TYPE "IOL_CONF"
// stored: IsFailsafeCompliant false
   STRUCT
      SELECTED : Struct
         SCRN_1 : Bool;   // SCREEN ONE SELECTED / SCREEN 1 SELECTED
         SCRN_2 : Bool;   // SCREEN TWO SELECTED / SCREEN 2 SELECTED
         SCRN_3 : Bool;   // SCREEN THREE SELECTED / SCREEN 3 SELECTED
         SCRN_4 : Bool;   // SCREEN FOUR SELECTED / SCREEN 4 SELECTED
         SCRN_5 : Bool;   // SCREEN FIVE SELECTED / SCREEN 5 SELECTED
         SCRN_6 : Bool;   // SCREEN SIX SELECTED / SCREEN 6 SELECTED
         SCRN_7 : Bool;   // SCREEN SEVEN SELECTED / SCREEN 7 SELECTED
         SCRN_8 : Bool;   // SCREEN EIGHT SELECTED / SCREEN 8 SELECTED
         SCRN_11 : Bool;   // SCREEN 11 SELECTED
         SCRN_12 : Bool;   // SCREEN 12 SELECTED
         SCRN_13 : Bool;   // SCREEN 13 SELECTED
         SCRN_14 : Bool;   // SCREEN 14 SELECTED
         SCRN_15 : Bool;   // SCREEN 15 SELECTED
         SCRN_16 : Bool;   // SCREEN 16 SELECTED
         SCRN_17 : Bool;   // SCREEN 17 SELECTED
         SCRN_18 : Bool;   // SCREEN 18 SELECTED
      END_STRUCT;
      HMI_VARIABLES : Struct
         DONE : Bool;   // HMI DONE BIT
         BUSY : Bool;   // HMI BUSY BIT
         ERROR : Bool;   // HMI ERROR BIT
         RD_WRT_HMI : Bool;   // HMI BUTTON READ/ WRITE SELECTION
         EXECUTE_ACTION : Bool;   // HMI EXECUTE READ/WRITE
         SPARE_205 : Bool;   // SPARE BIT
         SPARE_206 : Bool;   // SPARE BIT
         SPARE_207 : Bool;   // SPARE BIT
         SPARE_210 : Bool;   // SPARE BIT
         SPARE_211 : Bool;   // SPARE BIT
         SPARE_212 : Bool;   // SPARE BIT
         SPARE_213 : Bool;   // SPARE BIT
         SPARE_214 : Bool;   // SPARE BIT
         SPARE_215 : Bool;   // SPARE BIT
         SPARE_216 : Bool;   // SPARE BIT
         SPARE_217 : Bool;   // SPARE BIT
         IOL_LIST : Int;   // SELECTION LIST
         IO_LIST_OLD : Int;   // SELECTION LIST OLD
         SCRN_NMBR : Int;   // SELECTED SCREEN
         SCRN_NMBR_OLD : Int;   // SELECTED SCREEN OLD
         RND_INTRVL_1 : Real;   // ROUND INTERVAL FIRST VALUE
         RND_INTRVL_2 : Real;   // ROUND INTVERAL SECOND VALUE
         VAR_ERROR : Byte;   // VARIABLE NUMBER ERROR TAKE PLACE
         TOT_FLT : Byte;   // TOTAL FAULT
         FIRST_VALUE_DISPLAY : Real;   // HMI FIRST VALUE DISPLAY
         SECOND_VALUE_DISPLAY : Real;   // HMI SECOND VALUE DISPLAY
         SPARE_DISPLAY0 : Real;   // HMI SPARE DISPLAY
         SPARE_DISPLAY1 : Real;   // HMI SPARE DISPLAY
         SPARE_DISPLAY2 : Real;   // HMI SPARE DISPLAY
         REAL_VALUE : Array[0..17] of Real;   // REAL VALUE
      END_STRUCT;
      SPARE : Array[1..24] of Byte;
      GEOADR { ExternalAccessible := 'False'; ExternalVisible := 'False'; ExternalWritable := 'False'; S7_SetPoint := 'True'} : GEOADDR;   // INFO TO DETERMINE HW_IO
      CONFIG_DATA : Struct
         SPARE : UInt;   // DATA ADDRESS ID / Spare
         DATA_PORT : UInt;   // DATA PORT
         CAP_NMBR : UInt;   // CAP NUMBER
         VAR_RO : UInt;   // READ ONLY VARIABLES
         TOT_REAL_VAR : UInt;   // TOTAL REAL VARIABLES TO READ
         REAL_VAR_ARRAY_POS : UInt;   // REAL VARIABLES FIRST POSITION AT ARRAY
         TOT_VAR_TO_RD : UInt;   // TOTAL VARIABLES TO READ
      END_STRUCT;
      IOL_CONF : Array[1..20] of Struct
         INDX : Int;   // INDEX
         SBINDX : Int;   // SUBINDEX
         LNG : Int;   // LENGTH
         GRDNT : Real;   // GRADIENT
         OFFST : Real;   // OFFSET
         ROUND_1_OR_2 : Int;   // ROUND INTERVAL TO USE 1 OR 2
      END_STRUCT;
   END_STRUCT;
   // // GEOADR.HWTYPE : HW type (info to obtain from hw component) 4=module
   // // GEOADR.AREA : Normally not used
   // // GEOADR.IOSYSTEM : Network the IO master is on (100 profinet)(Normally always 100)
   // // GEOADR.STATION : Device No. of the IO master in hardware
   // // GEOADR.SLOT : Slot Number in hardware
   // // GEOADR.SUBSLOT : Sub Slot Number if necessary (Normally not used)
END_TYPE

TYPE "LIOLink_typeDiagnostics"
// stored: IsFailsafeCompliant false
   STRUCT
      status { ExternalVisible := 'False'; ExternalWritable := 'False'} : Word;   // Status of the Block or error identification when error occurred
      subfunctionStatus { ExternalVisible := 'False'; ExternalWritable := 'False'} : DWord;   // Status or return value of called FB's, FCs and system blocks
      stateNumber { ExternalVisible := 'False'; ExternalWritable := 'False'} : DInt;   // State in the state machine of the block where the error occurred
   END_STRUCT;
END_TYPE

TYPE "AXIS_MANAGEMENT"
// stored: IsFailsafeCompliant false
   STRUCT
      UNIT_01_HM_PSTN : Bool;   // UNIT 01 HOME POSITION
      UNIT_01_MAINT_POS : Bool;   // UNIT 01 MAINTENACE POSITION
      UNIT_01_ST1_OUT_OF_CLLSN_ST0 : Bool;   // UNIT 01 STATION 1 OUT OF COLLISION STATION 0
      UNIT_01_ST2_OUT_OF_CLLSN_ST0 : Bool;   // UNIT 01 STATION 2 OUT OF COLLISION STATION 0
      UNIT_01_ST3_OUT_OF_CLLSN_ST0 : Bool;   // UNIT 01 STATION 3 OUT OF COLLISION STATION 0
      UNIT_01_ST4_OUT_OF_CLLSN_ST0 : Bool;   // UNIT 01 STATION 4 OUT OF COLLISION STATION 0
      UNIT_01_ST3_AX_IN_HM_PSTN_XYZ : Bool;   // UNIT 01 STATION 3 AXIS IN HOME POSITION X-Y-Z
      UNIT_01_SPINDLES_STOP_AUX : Bool;   // UNIT 01 SPINDLES STOPPED AUXILIARY
      UNIT_01_MRPS_P_GG_RTN : Bool;   // UNIT 01 MARPOSS PLUG GAUGE RETURNED
      UNIT_01_IN_TL_POS : Bool;   // UNIT 01 IN TOOL POSITION
      UNIT_02_HM_PSTN : Bool;   // UNIT 02 HOME POSITION
      UNIT_02_MAINT_POS : Bool;   // UNIT 02 MAINTENACE POSITION
      UNIT_02_ST1_OUT_OF_CLLSN_ST0 : Bool;   // UNIT 02 STATION 1 OUT OF COLLISION STATION 0
      UNIT_02_ST2_OUT_OF_CLLSN_ST0 : Bool;   // UNIT 02 STATION 2 OUT OF COLLISION STATION 0
      UNIT_02_ST3_OUT_OF_CLLSN_ST0 : Bool;   // UNIT 02 STATION 3 OUT OF COLLISION STATION 0
      UNIT_02_ST4_OUT_OF_CLLSN_ST0 : Bool;   // UNIT 01 STATION 4 OUT OF COLLISION STATION 0
      UNIT_02_ST3_AX_IN_HM_PSTN_XYZ : Bool;   // UNIT 02 AXIS IN HOME POSITION X-Y-Z
      UNIT_02_SPINDLES_STOP_AUX : Bool;   // UNIT 02 SPINDLES STOPPED AUXILIARY
      UNIT_02_MRPSS_MSRG_PRB_RTN : Bool;   // UNIT 02 MARPOSS PLUG GAUGE RETURNED
      UNIT_02_IN_TL_POS : Bool;   // UNIT 02 IN TOOL POSITION
      UNIT_01_ST0_AX_E10_HM_PSTN : Bool;   // UNIT 01 STATION 0 AXIS E10 HOME POSITION
      UNIT_02_ST0_AX_E20_HM_PSTN : Bool;   // UNIT 02 STATION 0 AXIS E20 HOME POSITION
      FIXTURE_HM_PSTN : Bool;   // UNIT FIXTURE HOME POSITION
      FIXTURE_DBB70_0 : Bool;   // UNIT FIXTURE DBB70=0 (90)
      FIXTURE_DBB70_1 : Bool;   // UNIT FIXTURE DBB70=1 (-90)
      FIXTURE_1_LOAD_UNLOAD_POS : Bool;   // FIXTURE 1 IN LOAD UNLOAD POSITION (180)
      FIXTURE_2_LOAD_UNLOAD_POS : Bool;   // FIXTURE 2 IN LOAD UNLOAD POSITION (0)
      FIXTURE_1_MANUAL_LOAD_UNLOAD_POS : Bool;   // FIXTURE 1 IN MANUAL LOAD UNLOAD POSITION
      FIXTURE_2_MANUAL_LOAD_UNLOAD_POS : Bool;   // FIXTURE 2 IN MANUAL LOAD UNLOAD POSITION
      GENRL_RTN_CND_ALL_CLG_CYL_UNIT_01 : Bool;   // GENERAL RETURN CONDITIONS FOR ALL CLAMPING CYLINDERS UNIT 01
      GENRL_RTN_CND_ALL_CLG_CYL_UNIT_02 : Bool;   // GENERAL RETURN CONDITIONS FOR ALL CLAMPING CYLINDERS UNIT 02
      CH1_PRMR_SET_SLCTN_A : Bool;   // CHANNEL 1 PARAMETER SET SELECTION A
      CH2_PRMR_SET_SLCTN_A : Bool;   // CHANNEL 2 PARAMETER SET SELECTION A
      CH3_PRMR_SET_SLCTN_A : Bool;   // CHANNEL 3 PARAMETER SET SELECTION A
      CH4_PRMR_SET_SLCTN_A : Bool;   // CHANNEL 4 PARAMETER SET SELECTION A
      CH5_PRMR_SET_SLCTN_A : Bool;   // CHANNEL 5 PARAMETER SET SELECTION A
      CH6_PRMR_SET_SLCTN_A : Bool;   // CHANNEL 6 PARAMETER SET SELECTION A
      CH7_PRMR_SET_SLCTN_A : Bool;   // CHANNEL 7 PARAMETER SET SELECTION A
      CH8_PRMR_SET_SLCTN_A : Bool;   // CHANNEL 8 PARAMETER SET SELECTION A
      CH9_PRMR_SET_SLCTN_A : Bool;   // CHANNEL 9 PARAMETER SET SELECTION A
      CH10_PRMR_SET_SLCTN_A : Bool;   // CHANNEL 10 PARAMETER SET SELECTION A
      CH1_PRMR_SET_SLCTD_A : Bool;   // CHANNEL 1 PARAMETER SET SELECTED A
      CH2_PRMR_SET_SLCTD_A : Bool;   // CHANNEL 2 PARAMETER SET SELECTED A
      CH3_PRMR_SET_SLCTD_A : Bool;   // CHANNEL 3 PARAMETER SET SELECTED A
      CH4_PRMR_SET_SLCTD_A : Bool;   // CHANNEL 4 PARAMETER SET SELECTED A
      CH5_PRMR_SET_SLCTD_A : Bool;   // CHANNEL 5 PARAMETER SET SELECTED A
      CH6_PRMR_SET_SLCTD_A : Bool;   // CHANNEL 6 PARAMETER SET SELECTED A
      CH7_PRMR_SET_SLCTD_A : Bool;   // CHANNEL 7 PARAMETER SET SELECTED A
      CH8_PRMR_SET_SLCTD_A : Bool;   // CHANNEL 8 PARAMETER SET SELECTED A
      CH9_PRMR_SET_SLCTD_A : Bool;   // CHANNEL 9 PARAMETER SET SELECTED A
      CH10_PRMR_SET_SLCTD_A : Bool;   // CHANNEL 10 PARAMETER SET SELECTED A
   END_STRUCT;
END_TYPE

TYPE "FULL_DEPTH_CLADDING"
// stored: IsFailsafeCompliant false
   STRUCT
      FULL_DEPTH : Bool;   // FULL DEPTH / TOTAL FULL DEPTH
      FULL_DEPTH_STA_1 : Bool;   // FULL DEPTH 1 / FULL DEPTH STATION 1
      FULL_DEPTH_STA_2 : Bool;   // FULL DEPTH 2 / FULL DEPTH STATION 2
      FULL_DEPTH_STA_3 : Bool;   // FULL DEPTH 3 / FULL DEPTH STATION 3
      FULL_DEPTH_STA_4 : Bool;   // FULL DEPTH 4 / FULL DEPTH STATION 4
      FULL_DEPTH_STA_5 : Bool;   // FULL DEPTH 5 / FULL DEPTH STATION 5
      FULL_DEPTH_STA_6 : Bool;   // FULL DEPTH 6 / FULL DEPTH STATION 6
      FULL_DEPTH_STA_7 : Bool;   // FULL DEPTH 7 / FULL DEPTH STATION 7
      PART_REJECTED_FIXTURE : Bool;   // PART REJECTED FIXTURE 1 / PART REJECTED FIXTURE
      AUX_FULL_DEPTH_STA_1 : Bool;   // AUXILIARY FULL DEPTH 1 / AUXILIARY FULL DEPTH STATION 1
      AUX_FULL_DEPTH_STA_2 : Bool;   // AUXILIARY FULL DEPTH 2 / AUXILIARY FULL DEPTH STATION 2
      AUX_FULL_DEPTH_STA_3 : Bool;   // AUXILIARY FULL DEPTH 3 / AUXILIARY FULL DEPTH STATION 3
      AUX_FULL_DEPTH_STA_4 : Bool;   // AUXILIARY FULL DEPTH 4 / AUXILIARY FULL DEPTH STATION 4
      AUX_FULL_DEPTH_STA_5 : Bool;   // AUXILIARY FULL DEPTH 5 / AUXILIARY FULL DEPTH STATION 5
      AUX_FULL_DEPTH_STA_6 : Bool;   // AUXILIARY FULL DEPTH 6 / AUXILIARY FULL DEPTH STATION 6
      AUX_FULL_DEPTH_STA_7 : Bool;   // AUXILIARY FULL DEPTH 7 / AUXILIARY FULL DEPTH STATION 7
      AUX_FULL_DEPTH_STA_8 : Bool;   // AUXILIARY FULL DEPTH 8 / AUXILIARY FULL DEPTH STATION 8
      AUX_FULL_DEPTH_PULSE_STA_1 : Bool;   // AUXILIARY FULL DEPTH PULSE 1 / AUXILIARY FULL DEPTH PULSE STATION 1
      AUX_FULL_DEPTH_PULSE_STA_2 : Bool;   // AUXILIARY FULL DEPTH PULSE 2 / AUXILIARY FULL DEPTH PULSE STATION 2
      AUX_FULL_DEPTH_PULSE_STA_3 : Bool;   // AUXILIARY FULL DEPTH PULSE 3 / AUXILIARY FULL DEPTH PULSE STATION 3
      AUX_FULL_DEPTH_PULSE_STA_4 : Bool;   // AUXILIARY FULL DEPTH PULSE 4 / AUXILIARY FULL DEPTH PULSE STATION 4
      AUX_FULL_DEPTH_PULSE_STA_5 : Bool;   // AUXILIARY FULL DEPTH PULSE 5 / AUXILIARY FULL DEPTH PULSE STATION 5
      AUX_FULL_DEPTH_PULSE_STA_6 : Bool;   // AUXILIARY FULL DEPTH PULSE 6 / AUXILIARY FULL DEPTH PULSE STATION 6
      AUX_FULL_DEPTH_PULSE_STA_7 : Bool;   // AUXILIARY FULL DEPTH PULSE 7 / AUXILIARY FULL DEPTH PULSE STATION 7
      AUX_FULL_DEPTH_PULSE_STA_8 : Bool;   // AUXILIARY FULL DEPTH PULSE 8 / AUXILIARY FULL DEPTH PULSE STATION 8
      FD_PULSE : Bool;   // FULL DEPTH PULSE / TOTAL FULL DEPTH PULSE
      FD_STA_1_PULSE : Bool;   // FULL DEPTH 1 PULSE / FULL DEPTH STATION 1 PULSE
      FD_STA_2_PULSE : Bool;   // FULL DEPTH 2 PULSE / FULL DEPTH STATION 2 PULSE
      FD_STA_3_PULSE : Bool;   // FULL DEPTH 3 PULSE / FULL DEPTH STATION 3 PULSE
      FD_STA_4_PULSE : Bool;   // FULL DEPTH 4 PULSE / FULL DEPTH STATION 4 PULSE
      FD_STA_5_PULSE : Bool;   // FULL DEPTH 5 PULSE / FULL DEPTH STATION 5 PULSE
      FD_STA_6_PULSE : Bool;   // FULL DEPTH 6 PULSE / FULL DEPTH STATION 6 PULSE
      FD_STA_7_PULSE : Bool;   // FULL DEPTH 7 PULSE / FULL DEPTH STATION 7 PULSE
   END_STRUCT;
END_TYPE

TYPE "OPEN_CLOSE"
// stored: IsFailsafeCompliant false
   STRUCT
      CLOSED_PART_A_I : Bool;   // ADVANCED PART "A" INPUT / CLOSED PART A INPUT
      CLOSED_PART_B_I : Bool;   // ADVANCED PART "B" INPUT / CLOSED PART B INPUT
      CLOSED_PART_C_I : Bool;   // ADVANCED PART "C" INPUT / CLOSED PART C INPUT
      CLOSED_PART_D_I : Bool;   // ADVANCED PART "D" INPUT / CLOSED PART D INPUT
      CLOSED_PRESSURE_SW_1_I : Bool;   // ADVANCED PRESSURE SWITCH 1 / CLOSED PRESSURE SWITCH 1 INPUT
      CLOSED_PRESSURE_SW_2_I : Bool;   // ADVANCED PRESSURE SWITCH 2 / CLOSED PRESSURE SWITCH 2 INPUT
      OPEN_PART_A_I : Bool;   // RETURNED PART "A" INPUT / OPEN PART A INPUT
      OPEN_PART_B_I : Bool;   // RETURNED PART "B" INPUT / OPEN PART B INPUT
      OPEN_PART_C_I : Bool;   // RETURNED PART "C" INPUT / OPEN PART C INPUT
      OPEN_PART_D_I : Bool;   // RETURNED PART "D" INPUT / OPEN PART D INPUT
      OPEN_PRESSURE_SW_1_I : Bool;   // RETURNED PRESSURE SWITCH 1 / OPEN PRESSURE SWITCH 1 INPUT
      OPEN_PRESSURE_SW_2_I : Bool;   // RETURNED PRESSURE SWITCH 2 / OPEN PRESSURE SWITCH 2 INPUT
      CLOSED_LOW_PRESSURE_SW_I : Bool;   // CLOSED LOW PRESSURE SWITCH INPUT
      OPEN_LOW_PRESSURE_SW_I : Bool;   // OPEN LOW PRESSURE SWITCH INPUT
      ANY_CLOSED : Bool;   // ANY CLOSED INPUT
      ANY_OPEN : Bool;   // ANY OPEN INPUT
      GENERAL_CONDITIONS : Bool;   // GENERAL CONDITIONS
      CLOSE_CONDITIONS : Bool;   // ADVANCE CONDITIONS / CLOSE CONDITIONS
      OPEN_CONDITIONS : Bool;   // RETURN CONDITIONS / OPEN CONDITIONS
      RELEASE_PRESSURE_CONDITIONS : Bool;   // RELIEVE PRESSURE CONDITIONS / RELEASE PRESSURE CONDITIONS
      LOW_PRESSURE_CONDITIONS : Bool;   // RELIEVE PRESSURE CONDITIONS / LOW PRESSURE CONDITIONS
      GENERAL_CONDITIONS_HELP : Bool;   // GENERAL CONDITIONS HELP
      CLOSE_CONDITIONS_HELP : Bool;   // CLOSE CONDITIONS HELP
      OPEN_CONDITIONS_HELP : Bool;   // OPEN CONDITIONS HELP
      RELEASE_PRESSURE_CONDITIONS_HELP : Bool;   // RELEASE PRESSURE CONDITIONS HELP
      LOW_PRESSURE_CONDITIONS_HELP : Bool;   // LOW PRESSURE CONDITIONS HELP
      CLOSE_MANUAL_REQUEST : Bool;   // ADVANCE MANUAL REQUEST / CLOSE MANUAL REQUEST
      OPEN_MANUAL_REQUEST : Bool;   // RETURN MANUAL REQUEST / OPEN MANUAL REQUEST
      RELEASE_PRESSURE_MANUAL_REQUEST : Bool;   // RELIEVE PRESSURE MANUAL REQUEST / RELEASE PRESSURE MANUAL REQUEST
      LOW_PRESSURE_MANUAL_REQUEST : Bool;   // RELIEVE PRESSURE MANUAL REQUEST / LOW PRESSURE MANUAL REQUEST
      CLOSE_AUTO_REQUEST : Bool;   // ADVANCE AUTO REQUEST / CLOSE AUTO REQUEST
      OPEN_AUTO_REQUEST : Bool;   // RETURN AUTO REQUEST / OPEN AUTO REQUEST
      RELEASE_PRESSURE_AUTO_REQUEST : Bool;   // RELIEVE PRESSURE AUTO REQUEST / RELEASE PRESSURE AUTO REQUEST
      LOW_PRESSURE_AUTO_REQUEST : Bool;   // LOW PRESSURE AUTO REQUEST
      CLOSE_GLOBAL_REQUEST : Bool;   // ADVANCE GLOBAL REQUEST / CLOSE GLOBAL REQUEST
      OPEN_GLOBAL_REQUEST : Bool;   // RETURN GLOBAL REQUEST / OPEN GLOBAL REQUEST
      RELEASE_PRESSURE_GLOBAL_REQUEST : Bool;   // RELIEVE PRESSURE GLOBAL REQUEST / RELEASE PRESSURE GLOBAL REQUEST
      LOW_PRESSURE_GLOBAL_REQUEST : Bool;   // LOW PRESSURE GLOBAL REQUEST
      CLOSE_COMMAND : Bool;   // ADVANCE COMMAND / CLOSE COMMAND
      OPEN_COMMAND : Bool;   // RETURN COMMAND / OPEN COMMAND
      RELEASE_PRESSURE_COMMAND : Bool;   // RELIEVE PRESSURE COMMAND / RELEASE PRESSURE COMMAND
      CLOSE_LOW_PRESSURE_COMMAND : Bool;   // CLOSE LOW PRESSURE COMMAND
      OPEN_LOW_PRESSURE_COMMAND : Bool;   // OPEN LOW PRESSURE COMMAND
      CLOSE_LOW_PRESSURE : Bool;   // CLOSE LOW PRESSURE
      OPEN_LOW_PRESSURE : Bool;   // OPEN LOW PRESSURE
      FULL_CLOSED : Bool;   // ADVANCE / CLOSED AND COMMANDED
      FULL_OPEN : Bool;   // RETURN / OPEN AND COMMANDED
      FULL_LOW_PRESSURED : Bool;   // LOW PRESSURED AND COMMANDED
      CHECK_CLOSED : Bool;   // CHECK CLOSED AND COMMANDED
      CHECK_OPEN : Bool;   // CHECK OPEN AND COMMANDED
      CHECK_LOW_PRESSURED : Bool;   // CHECK LOW PRESSURED AND COMMANDED
      SIMULTANEITY_ALARM : Bool;   // SIMULTANEITY FAULT / SIMULTANEITY ALARM
      TIME_EXCEEDED_ALARM : Bool;   // TIME EXCEEDED / TIME EXCEEDED ALARM
      ANY_ACTIVE_ALARM : Bool;   // FAULT / ANY ACTIVE ALARM
      RHP_SEOC_ALARMS : Bool;   // RETURN HOME POSITION AND STOP END OF CYCLE ALARMS
      HMI_ACTD_LOW_AUX : Bool;   // HMI FLOWMETER SCREEN CLOSED LOW AUXILIARY
      HMI_DEACTD_LOW_AUX : Bool;   // HMI FLOWMETER SCREEN OPEN LOW AUXILIARY
      PULSE_1 : Bool;   // AUXILIAR ADVANCED PRESSURE SWITCH 1 FAULT / PULSE 1
      PULSE_2 : Bool;   // AUXILIAR ADVANCED PRESSURE SWITCH 2 FAULT / PULSE 2
      PULSE_3 : Bool;   // AUXILIAR RETURNED PRESSURE SWITCH 1 FAULT / PULSE 3
      PULSE_4 : Bool;   // AUXILIAR RETURNED PRESSURE SWITCH 2 FAULT / PULSE 4
      PULSE_5 : Bool;   // AUXILIAR RETURNED PRESSURE SWITCH 1 FAULT / PULSE 5
      PULSE_6 : Bool;   // AUXILIAR RETURNED PRESSURE SWITCH 2 FAULT / PULSE 6
      PULSE_7 : Bool;   // AUXILIAR RETURNED PRESSURE SWITCH 1 FAULT / PULSE 7
      PULSE_8 : Bool;   // AUXILIAR RETURNED PRESSURE SWITCH 2 FAULT / PULSE 8
   END_STRUCT;
END_TYPE

TYPE "ADVANCE_RETURN_CYL_CLADDING"
// stored: IsFailsafeCompliant false
   STRUCT
      GENERAL_CONDITIONS : Bool;   // GENERAL CONDITIONS
      ADVANCE_CONDITIONS : Bool;   // ADVANCE CONDITIONS
      RETURN_CONDITIONS : Bool;   // RETURN CONDITIONS
      GENERAL_CONDITIONS_HELP : Bool;   // GENERAL CONDITIONS HELP
      ADVANCE_CONDITIONS_HELP : Bool;   // ADVANCE CONDITIONS HELP
      RETURN_CONDITIONS_HELP : Bool;   // RETURN CONDITIONS HELP
      ADVANCE_HMI_REQUEST : Bool;   // ADVANCE HMI REQUEST / ADVANCE MANUAL HMI REQUEST
      RETURN_HMI_REQUEST : Bool;   // RETURN HMI REQUEST / RETURN MANUAL HMI REQUEST
      ADVANCE_MANUAL_REQUEST : Bool;   // ADVANCE MANUAL REQUEST
      RETURN_MANUAL_REQUEST : Bool;   // RETURN MANUAL REQUEST
      ADVANCE_AUTO_REQUEST : Bool;   // ADVANCE AUTO REQUEST
      RETURN_AUTO_REQUEST : Bool;   // RETURN AUTO REQUEST
      ADVANCE_GLOBAL_REQUEST : Bool;   // ADVANCE GLOBAL REQUEST
      RETURN_GLOBAL_REQUEST : Bool;   // RETURN GLOBAL REQUEST
      ADVANCE_COMMAND : Bool;   // ADVANCE COMMAND
      RETURN_COMMAND : Bool;   // RETURN COMMAND
      FULL_ADVANCED : Bool;   // ADVANCED FEEDBACK / ADVANCED AND COMMANDED
      FULL_RETURNED : Bool;   // RETURNED FEEDBACK / RETURNED AND COMMANDED
      SIMULTANEITY_ALARM : Bool;   // SIMULTANEITY FAULT / SIMULTANEITY ALARM
      TIME_EXCEEDED_ALARM : Bool;   // TIME EXCEEDED / TIME EXCEEDED ALARM
      ANY_ACTIVE_ALARM : Bool;   // FAULT / ANY ACTIVE ALARM
      IS_SEOC_ALARMS : Bool;   // INMEDIATE STOP AND STOP END OF CYCLE ALARMS
      PULSE_1 : Bool;   // PULSE 1
      PULSE_2 : Bool;   // PULSE 2
      PULSE_3 : Bool;   // PULSE 3
   END_STRUCT;
END_TYPE

TYPE "OPEN_CLOSE_HATCH_CLADDING"
// stored: IsFailsafeCompliant false
   STRUCT
      GENERAL_CONDITIONS : Bool;   // GENERAL CONDITIONS
      CLOSE_CONDITIONS : Bool;   // ADVANCE CONDITIONS / CLOSE CONDITIONS
      OPEN_CONDITIONS : Bool;   // RETURN CONDITIONS / OPEN CONDITIONS
      GENERAL_CONDITIONS_HELP : Bool;   // GENERAL CONDITIONS HELP
      CLOSE_CONDITIONS_HELP : Bool;   // CLOSE CONDITIONS HELP
      OPEN_CONDITIONS_HELP : Bool;   // OPEN CONDITIONS HELP
      CLOSE_HMI_REQUEST : Bool;   // ADVANCE HMI REQUEST / CLOSE MANUAL HMI REQUEST
      OPEN_HMI_REQUEST : Bool;   // RETURN HMI REQUEST / OPEN MANUAL HMI REQUEST
      CLOSE_MANUAL_REQUEST : Bool;   // ADVANCE MANUAL REQUEST / CLOSE MANUAL REQUEST
      OPEN_MANUAL_REQUEST : Bool;   // RETURN MANUAL REQUEST / OPEN MANUAL REQUEST
      CLOSE_AUTO_REQUEST : Bool;   // ADVANCE AUTO REQUEST / CLOSE AUTO REQUEST
      OPEN_AUTO_REQUEST : Bool;   // RETURN AUTO REQUEST / OPEN AUTO REQUEST
      CLOSE_GLOBAL_REQUEST : Bool;   // ADVANCE GLOBAL REQUEST / CLOSE GLOBAL REQUEST
      OPEN_GLOBAL_REQUEST : Bool;   // RETURN GLOBAL REQUEST / OPEN GLOBAL REQUEST
      CLOSE_COMMAND : Bool;   // ADVANCE COMMAND / CLOSE COMMAND
      OPEN_COMMAND : Bool;   // RETURN COMMAND / OPEN COMMAND
      FULL_CLOSED : Bool;   // ADVANCED FEEDBACK / CLOSED AND COMMANDED
      FULL_OPENED : Bool;   // RETURNED FEEDBACK / OPENED AND COMMANDED
      SIMULTANEITY_ALARM : Bool;   // SIMULTANEITY FAULT / SIMULTANEITY ALARM
      TIME_EXCEEDED_ALARM : Bool;   // TIME EXCEEDED / TIME EXCEEDED ALARM
      ANY_ACTIVE_ALARM : Bool;   // FAULT / ANY ACTIVE ALARM
      IS_SEOC_ALARMS : Bool;   // INMEDIATE STOP AND STOP END OF CYCLE ALARMS
      PULSE_1 : Bool;   // PULSE 1
      PULSE_2 : Bool;   // PULSE 2
      PULSE_3 : Bool;   // PULSE 3
   END_STRUCT;
END_TYPE

TYPE "SAFETY_BRAKE"
// stored: IsFailsafeCompliant false
   STRUCT
      GENERAL_CONDITIONS : Bool;   // GENERAL CONDITIONS
      BLOCK_CONDITIONS : Bool;   // BLOCK CONDITIONS
      UNBLOCK_CONDITIONS : Bool;   // UNBLOCK CONDITIONS
      GENERAL_CONDITIONS_HELP : Bool;   // GENERAL CONDITIONS HELP
      BLOCK_CONDITIONS_HELP : Bool;   // BLOCK CONDITIONS HELP
      UNBLOCK_CONDITIONS_HELP : Bool;   // UNBLOCK CONDITIONS HELP
      BLOCK_MANUAL_REQUEST : Bool;   // BLOCK MANUAL REQUEST
      UNBLOCK_MANUAL_REQUEST : Bool;   // UNBLOCK MANUAL REQUEST
      BLOCK_HMI_REQUEST : Bool;   // BLOCK HMI REQUEST
      UNBLOCK_HMI_REQUEST : Bool;   // UNBLOCK HMI REQUEST
      BLOCK_AUTO_REQUEST : Bool;   // BLOCK AUTO REQUEST
      UNBLOCK_AUTO_REQUEST : Bool;   // UNBLOCK AUTO REQUEST
      BLOCK_GLOBAL_REQUEST : Bool;   // BLOCK GLOBAL REQUEST
      UNBLOCK_GLOBAL_REQUEST : Bool;   // UNBLOCK GLOBAL REQUEST
      BLOCK_COMMAND : Bool;   // BLOCK COMMAND
      UNBLOCK_COMMAND : Bool;   // UNBLOCK COMMAND
      FULL_BLOCKED : Bool;   // BLOCK FEEDBACK / BLOCKED AND COMMANDED
      FULL_UNBLOCKED : Bool;   // UNBLOCK FEEDBACK / UNBLOCKED AND COMMANDED
      SIMULTANEITY_ALARM : Bool;   // SIMULTANEITY FAULT / SIMULTANEITY ALARM
      TIME_EXCEEDED_ALARM : Bool;   // TIME EXCEEDED / TIME EXCEEDED ALARM
      ANY_ACTIVE_ALARM : Bool;   // FAULT / ANY ACTIVE ALARM
      IS_SEOC_ALARMS : Bool;   // IMMEDIATE STOP AND STOP END OF CYCLE ALARMS
      PULSE_1 : Bool;   // PULSE 1
      PULSE_2 : Bool;   // PULSE 2
      PULSE_3 : Bool;   // PULSE 3
   END_STRUCT;
END_TYPE

TYPE "SAFETY_DOOR"
// stored: IsFailsafeCompliant false
   STRUCT
      CLOSED_I : Bool;   // CLOSED INPUT
      LOCKED_I : Bool;   // LOCKED INPUT
      OPEN_I : Bool;   // OPENED INPUT / OPEN INPUT
      UNLOCKED_I : Bool;   // UNLOCKED INPUT
      LOCK_GENERAL_CONDITIONS : Bool;   // LOCK GENERAL CONDITIONS
      LOCK_MANUAL_REQUEST : Bool;   // LOCK MANUAL REQUEST
      LOCK_HMI_REQUEST : Bool;   // LOCK SAFETY DOOR HMI REQUEST / LOCK HMI REQUEST
      LOCK_AUTO_REQUEST : Bool;   // LOCK AUTO REQUEST
      LOCK_GLOBAL_REQUEST : Bool;   // LOCK GLOBAL REQUEST
      LOCK_COMMAND : Bool;   // LOCK COMMAND
      LOCK : Bool;   // LOCK
      CLOSED_AND_LOCKED : Bool;   // CLOSED AND LOCKED
      UNLOCK_GENERAL_CONDITIONS : Bool;   // UNLOCK GENERAL CONDITIONS
      PARTIAL_UNLOCK_GENERAL_CONDITIONS : Bool;   // PARTIAL UNLOCK GENERAL CONDITIONS
      UNLOCK_MANUAL_REQUEST : Bool;   // UNLOCK MANUAL REQUEST
      UNLOCK_HMI_REQUEST : Bool;   // UNLOCK SAFETY DOOR HMI REQ / UNLOCK HMI REQUEST
      UNLOCK_AUTO_REQUEST : Bool;   // UNLOCK AUTO REQUEST
      UNLOCK_GLOBAL_REQUEST : Bool;   // UNLOCK GLOBAL REQUEST
      UNLOCK_COMMAND : Bool;   // UNLOCK COMMAND
      UNLOCK : Bool;   // UNLOCK
      OPEN_OR_UNLOCKED : Bool;   // OPENED AND UNLOCKED / OPEN OR UNLOCKED
      NOT_CLOSED_AND_LOCKED_ALARM : Bool;   // SAFETY DOOR FAULT / NOT CLOSED AND LOCKED ALARM
      DEPRESSURIZE_HYDRAULIC_DRIVE_ALARM : Bool;   // NOT POSSIBLE TO UNLOCK DEPRESSURIZE HYDRAULIC DRIVE ALARM
      NOT_CLOSED_AND_LOCKED_PREALARM : Bool;   // SAFE DOOR NOT CLOSED HELP / NOT CLOSED AND LOCKED WARNING
      UNLOCK_REQUEST_WARNING : Bool;   // UNLOCK REQUEST WARNING
      LOCK_GENERAL_CONDITIONS_HELP : Bool;   // LOCK GENERAL CONDITIONS HELP
      UNLOCK_GENERAL_CONDITIONS_HELP : Bool;   // UNLOCK GENERAL CONDITIONS HELP
      LOCK_MANUAL_REQUEST_AUX : Bool;   // AUXILIAR UNLOCK / LOCK MANUAL REQUEST AUXILIARY
      PARTIAL_UNLOCK_GENERAL_CONDITIONS_AUX : Bool;   // AUXILIAR UNLOCK / PARTIAL UNLOCK GENERAL CONDITIONS AUXILIARY
      UNLOCK_MANUAL_REQUEST_AUX : Bool;   // AUXILIAR UNLOCK / UNLOCK MANUAL REQUEST AUXILIARY
      UNLOCK_AUTO_REQUEST_AUX : Bool;   // AUXILIAR UNLOCK / UNLOCK AUTO REQUEST AUXILIARY
      UNLOCK_AUX : Bool;   // AUXILIAR UNLOCK / UNLOCK AUXILIARY
      PREALARM_GONE : Bool;   // AUXILIAR UNLOCK / WARNING GONE
      TIMER_PARTIAL_UNLOCK_GENERAL_CONDITIONS : TON_TIME;   // PARTIAL UNLOCK GENERAL CONDITIONS TIMER
      TIMER_UNLOCK : TON_TIME;   // UNLOCK TIMER
      TIMER_NOT_POSSIBLE_TO_UNLOCK : TON_TIME;   // NOT POSSIBLE TO UNLOCK TIMER
   END_STRUCT;
END_TYPE

TYPE "LAYOUT"
// stored: IsFailsafeCompliant false
   STRUCT
      Arrow : Array[0..79] of Bool;   // Arrow
      LED : Array[0..79] of Bool;   // LED
      Image : Array[0..79] of Bool;   // Image
      Text : Array[0..79] of Bool;   // Text
      IO_field : Array[0..79] of Bool;   // IO_field
      ProgressBar : Array[0..79] of Bool;   // ProgressBar
      Table0 : Bool;   // Table0
      Table1 : Bool;   // Table1
      Table2 : Bool;   // Table2
      Table3 : Bool;   // Table3
      Table4 : Bool;   // Table4
      Table5 : Bool;   // Table5
      Table6 : Bool;   // Table6
      Table7 : Bool;   // Table7
      Curve0 : Bool;   // Curve0
      Curve1 : Bool;   // Curve1
      Curve2 : Bool;   // Curve2
      Curve3 : Bool;   // Curve3
      Curve4 : Bool;   // Curve4
      Curve5 : Bool;   // Curve5
      Curve6 : Bool;   // Curve6
      Curve7 : Bool;   // Curve7
      Internet0 : Bool;   // Internet0
      Internet1 : Bool;   // Internet1
      Internet2 : Bool;   // Internet2
      Internet3 : Bool;   // Internet3
      Internet4 : Bool;   // Internet4
      Internet5 : Bool;   // Internet5
      Internet6 : Bool;   // Internet6
      Internet7 : Bool;   // Internet7
      SoftkeyLeft0 : Bool;   // SoftkeyLeft0
      SoftkeyLeft1 : Bool;   // SoftkeyLeft1
      SoftkeyLeft2 : Bool;   // SoftkeyLeft2
      SoftkeyLeft3 : Bool;   // SoftkeyLeft3
      SoftkeyLeft4 : Bool;   // SoftkeyLeft4
      SoftkeyLeft5 : Bool;   // SoftkeyLeft5
      SoftkeyLeftAll : Bool;   // SoftkeyLeftAll
      reserveleft : Bool;   // reserveleft
      SoftkeyRight0 : Bool;   // SoftkeyRight0
      SoftkeyRight1 : Bool;   // SoftkeyRight1
      SoftkeyRight2 : Bool;   // SoftkeyRight2
      SoftkeyRight3 : Bool;   // SoftkeyRight3
      SoftkeyRight4 : Bool;   // SoftkeyRight4
      SoftkeyRight5 : Bool;   // SoftkeyRight5
      SoftkeyRightAll : Bool;   // SoftkeyRightAll
      reserveright : Bool;   // reserveright
      Pushbutton0 : Bool;   // Pushbutton0
      Pushbutton1 : Bool;   // Pushbutton1
      Pushbutton2 : Bool;   // Pushbutton2
      Pushbutton3 : Bool;   // Pushbutton3
      Pushbutton4 : Bool;   // Pushbutton4
      Pushbutton5 : Bool;   // Pushbutton5
      Pushbutton6 : Bool;   // Pushbutton6
      Pushbutton7 : Bool;   // Pushbutton7
      Pushbutton8 : Bool;   // Pushbutton8
      Pushbutton9 : Bool;   // Pushbutton9
      Pushbutton10 : Bool;   // Pushbutton10
      Pushbutton11 : Bool;   // Pushbutton11
      Pushbutton12 : Bool;   // Pushbutton12
      Pushbutton13 : Bool;   // Pushbutton13
      Pushbutton14 : Bool;   // Pushbutton14
      Pushbutton15 : Bool;   // Pushbutton15
      Pushbutton16 : Bool;   // Pushbutton16
      Pushbutton17 : Bool;   // Pushbutton17
      Pushbutton18 : Bool;   // Pushbutton18
      Pushbutton19 : Bool;   // Pushbutton19
      Pushbutton20 : Bool;   // Pushbutton20
      Pushbutton21 : Bool;   // Pushbutton21
      Pushbutton22 : Bool;   // Pushbutton22
      Pushbutton23 : Bool;   // Pushbutton23
      Pushbutton24 : Bool;   // Pushbutton24
      Pushbutton25 : Bool;   // Pushbutton25
      Pushbutton26 : Bool;   // Pushbutton26
      Pushbutton27 : Bool;   // Pushbutton27
      Pushbutton28 : Bool;   // Pushbutton28
      Pushbutton29 : Bool;   // Pushbutton29
      Pushbutton30 : Bool;   // Pushbutton30
      Pushbutton31 : Bool;   // Pushbutton31
      byte69 : Byte;   // byte69
   END_STRUCT;
END_TYPE

TYPE "READ_CNC_MEMORY_1"
// stored: IsFailsafeCompliant false
   STRUCT
      Read : Bool;   // Lesen der Daten angefordert
      Busy : Bool;   // Aufruf SFC51 ist aktiv
      ListenId : Word;   // Listen-ID, die ausgelesen werden soll, alle Speicherbereiche (1, 3)
      ListenIndex : Word;   // Index fuer den Datensatz, hier Anwenderspeicher
      RetVal : Int;   // Returnwert fuerdas Auslesen des Anwender-Spechers
      SZL_HEADER : Struct
         LengthDataBlock : Word;   // Laenge eines Datensatzes
         CountDataBlock : Word;   // Anzahl vorhandener / gelesener Datensaetze
      END_STRUCT;
   END_STRUCT;
END_TYPE

TYPE "READ_CNC_MEMORY_2"
// stored: IsFailsafeCompliant false
   STRUCT
      Index : Word;   // Index, 1 = Arbeitsspeicher
      Code : Word;   // Speichertyp, 1 = RAM, 2 = FEPROM, 3 = RAM und FEPROM
      Size : DWord;   // Gesamtgroesse
      Mode : Word;   // Modus, Bit 0=RAM, 1=FEPROM, 2=RAM/FEPROM, 3=Code/Daten getr., 4=Code/Daten gem.
      Granu : Word;   // Immer 0
      Ber1 : DWord;   // Groesse des RAM's
      Occupied1 : DWord;   // Groesse des belegten RAM's
      Block1 : DWord;   // Groesster freier Block
      Ber2 : DWord;   // Groesse des FEPROM's
      Occupied2 : DWord;   // Groesse des belegten FEPROM's
      Block2 : DWord;   // Groesster frreier Block
   END_STRUCT;
END_TYPE

TYPE "READ_WRITE_DATA"
// stored: IsFailsafeCompliant false
   STRUCT
      IO_field : Array[0..79] of Bool;
      SoftkeyLeft0 : Bool;
      SoftkeyLeft1 : Bool;
      SoftkeyLeft2 : Bool;
      SoftkeyLeft3 : Bool;
      SoftkeyLeft4 : Bool;
      SoftkeyLeft5 : Bool;
      SoftkeyLeft6 : Bool;
      Page_up : Bool;
      SoftkeyRight0 : Bool;
      SoftkeyRight1 : Bool;
      SoftkeyRight2 : Bool;
      SoftkeyRight3 : Bool;
      SoftkeyRight4 : Bool;
      SoftkeyRight5 : Bool;
      SoftkeyRight6 : Bool;
      Page_Down : Bool;
      Pushbutton : Array[12..21] of Byte;
   END_STRUCT;
END_TYPE

TYPE "TOOL_LIFE_PLC"
// stored: IsFailsafeCompliant false
   STRUCT
      IS_ALARMS : Bool;   // IMMEDIATE STOP ALARMS
      IS_SEOC_ALARMS : Bool;   // IMMEDIATE STOP & STOP END OF CYCLE ALARMS / IMMEDIATE STOP AND STOP END OF CYCLE ALARMS
      RHP_ALARMS : Bool;   // RETURN HOME POSITION ALARMS
      RHP_SEOC_ALARMS : Bool;   // RETURN HOME POSITION & STOP END OF CYCLE ALARMS / RETURN HOME POSITION AND STOP END OF CYCLE ALARMS
      SEOC_ALARMS : Bool;   // STOP END OF CYCLE ALARMS
      IS_WARNING : Bool;   // IMMEDIATE STOP WARNING / IMMEDIATE STOP WARNINGS
      RHP_WARNING : Bool;   // RETURN HOME POSITION WARNING / RETURN HOME POSITION WARNINGS
      SEOC_WARNING : Bool;   // STOP END OF CYCLE WARNING / STOP END OF CYCLE WARNINGS
      WARNING : Bool;   // WARNING / WARNINGS
      HELP : Bool;   // HELP
      SPARE_11 : Bool;
      SPARE_12 : Bool;
      TOOL_PREALARM : Bool;   // TOOL PREALARM
      TOOL_ALARM : Bool;   // TOOL ALARM
      WARNING_GONE : Bool;   // WARNING GONE
      SPARE_16 : Bool;
      LIFE_EXPIRED_TOOL : Array[1..15] of Bool;   // LIFE EXPIRED TOOL
      SPARE_18 : Bool;
      SPARE_19 : Bool;
      LIFE_WARNING_TOOL : Array[1..15] of Bool;   // LIFE WARNING TOOL
      SPARE_21 : Bool;
      SPARE_22 : Bool;
      COUNTING_ENABLE : Bool;   // COUNTING ENABLE
      COUNTIN_ENABLE_PULSE : Bool;   // COUNTING ENABLE PULSE
      SPARE_25 : Bool;
      SPARE_26 : Bool;
      SPARE_27 : Bool;
      SPARE_28 : Bool;
      SPARE_29 : Bool;
      SPARE_30 : Bool;
   END_STRUCT;
END_TYPE

TYPE "INTERLOCKS_ETXETAR_ROBOT_CELL_GENERAL"
// stored: IsFailsafeCompliant false
   STRUCT
      MACHINE_TO_CELL : Struct
         MCH_MEAS_STA_CALIBRATION_REQ : Bool;   // MACHINE MEAS STATION CALIBRATION REQUIRED
         MCH_MEAS_STA_READY_TO_MEASURE : Bool;   // MACHINE MEAS STATION READY TO MEASURE
         MCH_MEAS_STA_MEASURE_IN_PRCESS : Bool;   // MACHINE MEAS STATION MEASUREMENT IN PROCESS
         MCH_MEAS_STA_MEASURE_FINISHED : Bool;   // MACHINE MEAS STATION MEASUREMENT FINISHED
         MCH_MEAS_STA_HOME_POSITION : Bool;   // MACHINE MEAS STATION AT HOME POSITION
         MCH_MEAS_STA_FAULT : Bool;   // MACHINE MEAS STATION FAULT
         PNEUMATIC_IN_SERVICE_SPARE_0_5 : Bool;
         SPARE_0_7 : Bool;
         MCH_MEAS_STA_MICROEPSILON_FACE_R_ENABLED : Bool;   // MACHINE MEAS STATION MICROEPSILON FACE R ENABLED
         MCH_MEAS_STA_MICROEPSILON_FACE_N_ENABLED : Bool;   // MACHINE MEAS STATION MICROEPSILON FACE N ENABLED
         SPARE_1_2 : Bool;
         SPARE_1_3 : Bool;
         SPARE_1_4 : Bool;
         SPARE_1_5 : Bool;
         SPARE_1_6 : Bool;
         SPARE_1_7 : Bool;
         SPARE_MEAS_STA : Array[0..5] of Byte;
         COOLING_SPARE : Bool;
         SPARE_8_1 : Bool;
         SPARE_8_2 : Bool;
         SPARE_8_3 : Bool;
         SPARE_8_4 : Bool;
         SPARE_8_5 : Bool;
         SPARE_8_6 : Bool;
         SPARE_8_7 : Bool;
         SPARE_9_0 : Bool;
         SPARE_9_1 : Bool;
         SPARE_9_2 : Bool;
         SPARE_9_3 : Bool;
         SPARE_9_4 : Bool;
         SPARE_9_5 : Bool;
         SPARE_9_6 : Bool;
         SPARE_9_7 : Bool;
         SPARE_COOLING : Array[0..5] of Byte;
         MCH_EKS_CURRENT_PROTECTION_LVL : Byte;   // MACHINE EKS CURRENT ACCESS LEVEL
         MCH_EKS_IDENT_1 : Byte;   // MACHINE EKS OPERATOR ID CHAR 1
         MCH_EKS_IDENT_2 : Byte;   // MACHINE EKS OPERATOR ID CHAR 2
         MCH_EKS_IDENT_3 : Byte;   // MACHINE EKS OPERATOR ID CHAR 3
         MCH_EKS_IDENT_4 : Byte;   // MACHINE EKS OPERATOR ID CHAR 4
         MCH_EKS_IDENT_5 : Byte;   // MACHINE EKS OPERATOR ID CHAR 5
         MCH_EKS_IDENT_6 : Byte;   // MACHINE EKS OPERATOR ID CHAR 6
         MCH_EKS_IDENT_7 : Byte;   // MACHINE EKS OPERATOR ID CHAR 7
         MCH_EKS_IDENT_8 : Byte;   // MACHINE EKS OPERATOR ID CHAR 8
         MCH_EKS_OPERATOR_IDENTIFICATION : Byte;   // MACHINE EKS OPERATOR IDENTIFICATION
         SPARE_26_0 : Bool;
         SPARE_26_1 : Bool;
         SPARE_26_2 : Bool;
         SPARE_26_3 : Bool;
         SPARE_26_4 : Bool;
         SPARE_26_5 : Bool;
         SPARE_26_6 : Bool;
         SPARE_26_7 : Bool;
         SPARE_27_0 : Bool;
         SPARE_27_1 : Bool;
         SPARE_27_2 : Bool;
         SPARE_27_3 : Bool;
         SPARE_27_4 : Bool;
         SPARE_27_5 : Bool;
         SPARE_27_6 : Bool;
         SPARE_27_7 : Bool;
         SPARE_GENERAL : Array[0..34] of Byte;
      END_STRUCT;
      CELL_TO_MACHINE : Struct
         CELL_MEAS_STA_START_MEAS_CYCLE : Bool;   // CELL MEASURING STATION START MEASURING CYCLE
         CELL_MEAS_STA_START_CALIB_CYCLE : Bool;   // CELL MEASURING STATION START CALIBRATION CYCLE
         CELL_MEAS_STA_HOME_REQ : Bool;   // CELL MEASURING STATION HOME REQUEST
         CELL_MEAS_STA_FAULT : Bool;   // CELL MEASURING STATION FAULT
         CELL_MEAS_STA_RESET : Bool;   // CELL MEASURING STATION RESET
         CALIB_MODE_SLCTD_SPARE_0_5 : Bool;
         SPARE_0_6 : Bool;
         SPARE_0_7 : Bool;
         CELL_MEAS_STA_PART_LOADED : Bool;   // CELL MEASURING STATION PART LOADED
         CELL_MEAS_STA_PART_UNLOADED : Bool;   // CELL MEASURING STATION PART UNLOADED
         SPARE_1_2 : Bool;
         SPARE_1_3 : Bool;
         SPARE_1_4 : Bool;
         SPARE_1_5 : Bool;
         SPARE_1_6 : Bool;
         SPARE_1_7 : Bool;
         SPARE_MEAS_STA : Array[0..5] of Byte;
         CELL_COOLING_DEGRADED_MODE : Bool;   // CELL COOLING DEGRADED MODE
         SPARE_8_1 : Bool;
         SPARE_8_2 : Bool;
         SPARE_8_3 : Bool;
         SPARE_8_4 : Bool;
         SPARE_8_5 : Bool;
         SPARE_8_6 : Bool;
         SPARE_8_7 : Bool;
         SPARE_9_0 : Bool;
         SPARE_9_1 : Bool;
         SPARE_9_2 : Bool;
         SPARE_9_3 : Bool;
         SPARE_9_4 : Bool;
         SPARE_9_5 : Bool;
         SPARE_9_6 : Bool;
         SPARE_9_7 : Bool;
         SPARE_COOLING : Array[0..5] of Byte;
         CELL_STARVED : Bool;   // CELL STARVED
         CELL_BLOCKED : Bool;   // CELL BLOCKED
         SPARE_16_2 : Bool;
         SPARE_16_3 : Bool;
         SPARE_16_4 : Bool;
         SPARE_16_5 : Bool;
         SPARE_16_6 : Bool;
         SPARE_16_7 : Bool;
         SPARE_17_0 : Bool;
         SPARE_17_1 : Bool;
         SPARE_17_2 : Bool;
         SPARE_17_3 : Bool;
         SPARE_17_4 : Bool;
         SPARE_17_5 : Bool;
         SPARE_17_6 : Bool;
         SPARE_17_7 : Bool;
         SPARE_GENERAL : Array[0..45] of Byte;
      END_STRUCT;
   END_STRUCT;
END_TYPE

TYPE "INTERLOCKS_ETXETAR_ROBOT_CELL_PER_UNIT"
// stored: IsFailsafeCompliant false
   STRUCT
      MACHINE_TO_ROBOT : Struct
         MCH_HEARTBEAT : Bool;   // MACHINE HEARTBEAT (MACHINE TO GANTRY) / MACHINE HEARTBEAT
         MCH_E_STOP_OK : Bool;   // MACHINE EMERGENCY STOP OK (MACHINE TO GANTRY) / MACHINE EMERGENCY STOP OK
         MCH_FAULT : Bool;   // MACHINE FAULT PRESENT
         MCH_SAFETY_DOORS_CLSD_LCKD : Bool;   // MACHINE SAFETY GATES OK (LOCKED)(MACHINE TO GANTRY) / MACHINE SAFETY DOORS CLOSED AND LOCKED
         SPARE_0_4 : Bool;
         SPARE_0_5 : Bool;
         MCH_MANUAL_MODE : Bool;   // MACHINE IN MANUAL MODE (MACHINE TO GANTRY) / MACHINE MANUAL MODE SELECTED
         MCH_AUTO_MODE : Bool;   // MACHINE IN AUTO MODE(MACHINE TO GANTRY) / MACHINE AUTO MODE SELECTED
         MCH_AUTO_CYCLE_RUN : Bool;   // MACHINE AUTO CYCLE RUNNING (MACHINE TO GANTRY) / MACHINE CYCLE RUNNING IN AUTOMATIC MODE
         MCH_WARM_UP_CYCLE_RUN : Bool;   // MACHINE IS IN WARMUP CYCLE (MACHINE TO GANTRY) / MACHINE WARM UP CYCLE RUNNING
         MCH_RUN_OUT_CYCLE : Bool;   // MACHINE IN RUN OUT MODE (MACHINE TO GANTRY) / MACHINE RUN OUT CYCLE SELECTED
         MCH_CALIBRATION_CYCLE : Bool;   // MACHINE CALIBRATION CYCLE SELECTED
         MCH_MASTER_MEASUREMENT_CYCLE : Bool;   // MACHINE MASTER MEASUREMENT CYCLE SELECTED
         MCH_PART_DEMAND_SOON : Bool;   // MACHINE PART DEMAND SOON (MACHINE TO GANTRY) / MACHINE PART DEMAND SOON
         MCH_SAFETY_DOOR_OPEN_REQ : Bool;   // MACHINE SAFETY DOOR OPEN REQUEST
         MCH_CELL_SAFETY_DOOR_OK_TO_OPEN : Bool;   // MACHINE APPROVAL TO OPEN THE CELL SAFETY DOOR
         MCH_EMPTY : Bool;   // MACHINE EMPTY
         MCH_FIX_1_ENABLED : Bool;   // MACHINE FIXTURE 1 ENABLED FOR LOAD/UNLOAD
         MCH_FIX_2_ENABLED : Bool;   // MACHINE FIXTURE 2 ENABLED FOR LOAD/UNLOAD
         MCH_FIX_3_ENABLED : Bool;   // MACHINE FIXTURE 3 ENABLED FOR LOAD/UNLOAD
         MCH_FIX_4_ENABLED : Bool;   // MACHINE FIXTURE 4 ENABLED FOR LOAD/UNLOAD
         MCH_FIX_1_PART_PRSNT : Bool;   // MACHINE FIXTURE 1 PART PRESENT
         MCH_FIX_2_PART_PRSNT : Bool;   // MACHINE FIXTURE 2 PART PRESENT
         MCH_FIX_3_PART_PRSNT : Bool;   // MACHINE FIXTURE 3 PART PRESENT
         MCH_FIX_4_PART_PRSNT : Bool;   // MACHINE FIXTURE 4 PART PRESENT
         MCH_FIX_1_CALIBRATION_REQ : Bool;   // MACHINE FIXTURE 1 CALIBRATION REQUIRED
         MCH_FIX_2_CALIBRATION_REQ : Bool;   // MACHINE FIXTURE 2 CALIBRATION REQUIRED
         MCH_FIX_3_CALIBRATION_REQ : Bool;   // MACHINE FIXTURE 3 CALIBRATION REQUIRED
         MCH_FIX_4_CALIBRATION_REQ : Bool;   // MACHINE FIXTURE 4 CALIBRATION REQUIRED
         SPARE_3_5 : Bool;
         SPARE_3_6 : Bool;
         SPARE_3_7 : Bool;
         CLEAR_LOAD_UNLOAD : Bool;   // MACHINE PART TYPE CHANGE IS POSSIBLE (MACHINE TO GANTRY) / MACHINE CLEAR TO LOAD / UNLOAD PARTS
         MCH_UNLOAD_REQUEST_FACE_R : Bool;   // MACHINE UNLOAD REQUEST FACE R
         MCH_UNLOAD_REQUEST_FACE_N : Bool;   // MACHINE UNLOAD REQUEST FACE N
         MCH_LOAD_REQUEST_FACE_R : Bool;   // MACHINE LOAD REQUEST FACE R
         MCH_LOAD_REQUEST_FACE_N : Bool;   // MACHINE SUSPECT PART FROM MACHINE (MACHINE TO GANTRY) / MACHINE LOAD REQUEST FACE N
         MCH_UNLD_ANTICIPATION_FACE_R : Bool;   // MACHINE EMPTY (MACHINE TO GANTRY) / MACHINE UNLOAD ANTICIPATION FACE R
         MCH_UNLD_ANTICIPATION_FACE_N : Bool;   // MACHINE UNLOAD ANTICIPATION FACE N
         MCH_LOAD_ANTICIPATION_FACE_R : Bool;   // MACHINE QUALITY CHECK WARNING (MACHINE TO GANTRY) / MACHINE LOAD ANTICIPATION FACE R
         MCH_LOAD_ANTICIPATION_FACE_N : Bool;   // MACHINE QUALITY CHECK FAULT (MACHINE TO GANTRY) / MACHINE LOAD ANTICIPATION FACE N
         MCH_PART_A_PRESENT : Bool;   // MACHINE QUALITY CHECK FAULT (MACHINE TO GANTRY) / MACHINE PART A PRESETN
         MCH_PART_A_MACHINED : Bool;   // MACHINE QUALITY CHECK FAULT (MACHINE TO GANTRY) / MACHINE PART A MACHINED
         MCH_PART_A_REJECTED : Bool;   // MACHINE QUALITY CHECK ACKNOWLEDGED (MACHINE TO GANTRY) / MACHINE PART A REJECTED
         MCH_PART_A_QUALITY : Bool;   // MACHINE PART A QUALITY
         SPARE_5_5 : Bool;   // MACHINE READY TO ACCEPT REWORK PART (MACHINE TO GANTRY)
         SPARE_5_6 : Bool;
         SPARE_5_7 : Bool;
         SPARE_6_0 : Bool;   // MACHINE CLEAR TO LOAD/UNLOAD (MACHINE TO GANTRY)
         SPARE_6_1 : Bool;   // MACHINE READY TO UNLOAD PART (MACHINE TO GANTRY)
         SPARE_6_2 : Bool;   // MACHINE READY TO LOAD PART (MACHINE TO GANTRY)
         SPARE_6_3 : Bool;   // MACHINE PART PRESENT (MACHINE TO GANTRY)
         SPARE_6_4 : Bool;   // MACHINE GOOD PART (MACHINE TO GANTRY)
         SPARE_6_5 : Bool;
         SPARE_6_6 : Bool;
         SPARE_6_7 : Bool;
         MCH_PART_TYPE : Byte;   // MACHINE PART IS CLAMPED (MACHINE TO GANTRY) / MACHINE PART TYPE
         SPARE : Array[0..55] of Byte;
      END_STRUCT;
      ROBOT_TO_MACHINE : Struct
         RBT_HEARTBEAT : Bool;   // GANTRY HEARTBEAT (GANTRY TO MACHINE) / ROBOT HEARTBEAT
         RBT_E_STOP_OK : Bool;   // GANTRY EMERGENCY STOP OK (GANTRY TO MACHINE) / ROBOT EMERGENCY STOP OK
         RBT_FAULT : Bool;   // ROBOT FAULT PRESENT
         RBT_SAFETY_DOOR_CLSD_LCKD : Bool;   // ROBOT SAFETY DOOR CLOSED AND LOCKED
         RBT_CELL_EMPTY : Bool;   // ROBOT CELL EMPTY
         SPARE_0_5 : Bool;
         SPARE_0_6 : Bool;
         SPARE_0_7 : Bool;
         RBT_MANUAL_MODE : Bool;   // GANTRY IN MANUAL MODE (GANTRY TO MACHINE) / ROBOT MANUAL MODE SELECTED
         RBT_AUTO_MODE : Bool;   // GANTRY IN AUTO MODE (GANTRY TO MACHINE) / ROBOT AUTO MODE SELECTED
         RBT_AUTO_CYCLE_RUN : Bool;   // GANTRY IN AUTO CYCLE RUNNING (GANTRY TO MACHINE) / ROBOT CYCLE RUNNING IN AUTOMATIC MODE
         SPARE_1_3 : Bool;   // GANTRY OVERHEAD DOOR CLOSED & LOCKED (GANTRY TO MACHINE)
         RBT_RUN_OUT_REQ : Bool;   // GANTRY PART TYPE CHANGE REQUESTED (GANTRY TO MACHINE) / ROBOT MACHINE RUN OUT REQUEST
         RBT_RUN_OUT_COMPLETED : Bool;   // GANTRY IN RUN OUT COMPLETE(GANTRY TO MACHINE) / ROBOT RUN OUT COMPLETED
         RBT_SAFETY_DOOR_OPEN_REQ : Bool;   // ROBOT ANY CELL SAFETY DOOR OPEN REQUEST
         RBT_MCH_SAFETY_DOOR_OK_TO_OPEN : Bool;   // ROBOT APPROVAL TO OPEN THE MACHINE SAFETY DOOR
         RBT_READY_TO_SERVICE : Bool;   // ROBOT IS READY TO SERVICE THE MACHINE
         RBT_OUT_OF_COLLISION_MACHINE : Bool;   // GANTRY CLEAR OF MACHINE (GANTRY TO MACHINE) / ROBOT OUT OF COLLISION MACHINE
         RBT_OUT_OF_COLLISION_FIXTURE : Bool;   // GANTRY CLEAR OF FIXTURE (GANTRY TO MACHINE) / ROBOT OUT OF COLLISION FIXTURE
         SPARE_2_3 : Bool;
         SPARE_2_4 : Bool;
         SPARE_2_5 : Bool;
         SPARE_2_6 : Bool;
         SPARE_2_7 : Bool;
         SPARE_3_0 : Bool;
         SPARE_3_1 : Bool;
         SPARE_3_2 : Bool;
         SPARE_3_3 : Bool;
         SPARE_3_4 : Bool;
         SPARE_3_5 : Bool;
         SPARE_3_6 : Bool;
         SPARE_3_7 : Bool;
         RBT_PART_ENABLED : Bool;   // ROBOT PART ENABLED
         SPARE_4_1 : Bool;   // GANTRY READY TO SERVICE MACHINE (GANTRY TO MACHINE)
         RBT_PART_FACE_R_TO_DELIVER : Bool;   // ROBOT PART FACE R TO DELIVER IMMEDIATELY
         RBT_PART_FACE_N_TO_DELIVER : Bool;   // ROBOT PART FACE N TO DELIVER IMMEDIATELY
         RBT_OUT_OF_PARTS_FACE_R_TO_DELIVER : Bool;   // ROBOT OUT OF PARTS FACE R IN CELL TO DELIVER
         RBT_OUT_OF_PARTS_FACE_N_TO_DELIVER : Bool;   // ROBOT OUT OF PARTS FACE N IN CELL TO DELIVER
         SPARE_4_6 : Bool;
         SPARE_4_7 : Bool;
         RBT_PART_LOADED : Bool;   // ROBOT PART LOADED
         RBT_PART_UNLOADED : Bool;   // ROBOT PART UNLOADED
         SPARE_5_2 : Bool;
         SPARE_5_3 : Bool;
         RBT_FIX_SKIP_REQ : Bool;   // ROBOT FIXTURE SKIP REQUEST
         SPARE_5_5 : Bool;
         SPARE_5_6 : Bool;
         SPARE_5_7 : Bool;
         RBT_PART_TYPE_REQ : Bool;   // ROBOT PART TYPE CHANGE REQUEST
         SPARE_6_1 : Bool;
         SPARE_6_2 : Bool;
         SPARE_6_3 : Bool;
         SPARE_6_4 : Bool;   // GANTRY ROUGH PART IS REWORK PART (GANTRY TO MACHINE)
         SPARE_6_5 : Bool;
         SPARE_6_6 : Bool;
         SPARE_6_7 : Bool;
         RBT_PART_TYPE : Byte;   // ROBOT PART TYPE
         SPARE : Array[0..55] of Byte;
      END_STRUCT;
   END_STRUCT;
END_TYPE

TYPE "LOAD_UNLOAD_ETXETAR_ROBOT_CELL"
// stored: IsFailsafeCompliant false
   STRUCT
      FROM_ROBOT_CELL : Struct
         PART_A_LOADED : Bool;   // PART 1 LOADED ARM 1 / PART A LOADED 1
         PART_A_UNLOADED : Bool;   // PART 1 UNLOADED ARM 1 / PART A UNLOADED 1
         PART_A_LOADED_P : Bool;   // PART 1 LOADED ARM 1 PULSE / PART A LOADED 1 PULSE
         PART_A_UNLOADED_P : Bool;   // PART 1 UNLOADED ARM 1 PULSE / PART A UNLOADED 1 PULSE
      END_STRUCT;
      TO_ROBOT_CELL : Struct
         REQ_LOAD_PART_A : Bool;   // REQUEST LOAD PART 1 ARM 1 / REQUEST LOAD PART A-1
         REQ_UNLOAD_PART_A : Bool;   // REQUEST UNLOAD PART 1 ARM 1 / REQUEST UNLOAD PART A-1
      END_STRUCT;
   END_STRUCT;
END_TYPE

TYPE "PART_ID"
// stored: IsFailsafeCompliant false
   STRUCT
      PART_ID : Array[0..63] of Byte;
   END_STRUCT;
END_TYPE

TYPE "QUALITY_CHECK"
// stored: IsFailsafeCompliant false
   STRUCT
      ACTUAL_COUNTER : Int;   // ACTUAL COUNTER
      PREALARM_COUNTER : Int;   // PREALARM COUNTER
      ALARM_COUNTER : Int;   // ALARM COUNTER
      INSPECTION : Bool;   // INSPECTION
      INSPECTION_EXPIRED : Bool;   // INSPECTION EXPIRED
      INSPECTION_PULSE : Bool;   // INSPECTION PULSE
      NOK : Bool;   // NOK
      OK : Bool;   // OK
      INSPECTION_ALARM_PULSE : Bool;   // INSPECTION ALARM PULSE
      INSPECTION_PULSE_AUX : Bool;   // INSPECTION PULSE AUX
      PULASE_AUX_QUALITY : Bool;   // PULASE AUX QUALITY
      QUALITY_COLOR : Byte;   // QUALITY COLOR
   END_STRUCT;
END_TYPE

TYPE "PART_STATUS_CLADDING"
// stored: IsFailsafeCompliant false
   STRUCT
      STATUS : Struct   // PART STATUS
         PRESENT : Bool;   // PART PRESENT
         OK : Bool;   // PART OK
         PART_REJECTED : Bool;   // PART REJECTED
         QUALITY_PART : Bool;   // PART QUALITY
         FULL_DEPTH : Bool;   // FULL DEPTH / PART FULL DEPTH
         MASTER_PART : Bool;   // MASTER PART / PART MASTER PART
         VIRTUAL_PART : Bool;   // PART VIRTUAL PART
         PART_TYPE : Byte;   // PART TYPE
         PART_MAIN_STATUS_COLOR : Int;   // PART MAIN STATUS HMI COLOR
         PART_CELL_STATUS_COLOR : Int;   // PART CELL STATUS HMI COLOR
         QUALITY_CHECK_STATUS : Struct
            PART_ON_DEMAND : Bool;   // PART QUALITY PART ON DEMAND
            TOOL_CHANGED : Bool;   // PART QUALITY TOOL CHANGED
            PART_TYPE_CHANGED : Bool;   // PART QUALITY PART TYPE CHANGED
            FIRST_CYCLE : Bool;   // PART QUALITY CHECK CYCLE INTERRUMPED
            SPARE : Byte;
         END_STRUCT;
         UNIT_01_STATUS : Struct
            PROCESSED_IN_F1 : Bool;   // PART UNIT 01 PROCESSED IN FIXTURE 1
            PROCESSED_IN_F2 : Bool;   // PART UNIT 01 PROCESSED IN FIXTURE 2
            PROCESSED_IN_F3 : Bool;   // PART UNIT 01 PROCESSED IN FIXTURE 3
            PROCESSED_IN_F4 : Bool;   // PART UNIT 01 PROCESSED IN FIXTURE 4
            FACE_R_STATION_1_DONE : Bool;   // PART UNIT 01 FACE R STATION 1 DONE
            FACE_R_STATION_2_DONE : Bool;   // PART UNIT 01 FACE R STATION 2 DONE
            FACE_R_STATION_3_DONE : Bool;   // PART UNIT 01 FACE R STATION 3 DONE
            FACE_R_STATION_4_DONE : Bool;   // PART UNIT 01 FACE R STATION 4 DONE
            FACE_N_STATION_1_DONE : Bool;   // PART UNIT 01 FACE N STATION 1 DONE
            FACE_N_STATION_2_DONE : Bool;   // PART UNIT 01 FACE N STATION 2 DONE
            FACE_N_STATION_3_DONE : Bool;   // PART UNIT 01 FACE N STATION 3 DONE
            FACE_N_STATION_4_DONE : Bool;   // PART UNIT 01 FACE N STATION 4 DONE
         END_STRUCT;
         UNIT_02_STATUS : Struct
            PROCESSED_IN_F1 : Bool;   // PART UNIT 02 PROCESSED IN FIXTURE 1
            PROCESSED_IN_F2 : Bool;   // PART UNIT 02 PROCESSED IN FIXTURE 2
            PROCESSED_IN_F3 : Bool;   // PART UNIT 02 PROCESSED IN FIXTURE 3
            PROCESSED_IN_F4 : Bool;   // PART UNIT 02 PROCESSED IN FIXTURE 4
            FACE_R_STATION_1_DONE : Bool;   // PART UNIT 02 FACE R STATION 1 DONE
            FACE_R_STATION_2_DONE : Bool;   // PART UNIT 02 FACE R STATION 2 DONE
            FACE_R_STATION_3_DONE : Bool;   // PART UNIT 02 FACE R STATION 3 DONE
            FACE_R_STATION_4_DONE : Bool;   // PART UNIT 02 FACE R STATION 4 DONE
            FACE_N_STATION_1_DONE : Bool;   // PART UNIT 02 FACE N STATION 1 DONE
            FACE_N_STATION_2_DONE : Bool;   // PART UNIT 02 FACE N STATION 2 DONE
            FACE_N_STATION_3_DONE : Bool;   // PART UNIT 02 FACE N STATION 3 DONE
            FACE_N_STATION_4_DONE : Bool;   // PART UNIT 02 FACE N STATION 4 DONE
         END_STRUCT;
         CELL_STATUS : Struct
            NEW : Bool;   // PART NEW
            NEW_CAMARA_OK : Bool;   // PART NEW CAMARA OK
            NEW_IN_TRANSIT : Bool;   // PART NEW IN TRANSIT
            U01_ONE_FACE_DONE : Bool;   // PART UNIT 01 ONE FACE DONE
            U01_ONE_FACE_DONE_ROTATED : Bool;   // PART UNIT 01 ONE FACE DONE ROTATED
            U01_DONE : Bool;   // PART UNIT 01 BOTH FACES DONE
            U01_DONE_IN_TRANSIT : Bool;   // PART UNIT 01 DONE IN TRANSIT
            U02_ONE_FACE_DONE : Bool;   // PART UNIT 02 ONE FACE DONE
            U02_ONE_FACE_DONE_IN_TRANSIT : Bool;   // PART UNIT 02 ONE FACE DONE IN TRANSIT
            U02_ONE_FACE_DONE_ROTATED : Bool;   // PART UNIT 02 ONE FACE DONE ROTATED
            U02_DONE : Bool;   // PART UNIT 02 BOTH FACES DONE
            U02_DONE_IN_TRANSIT : Bool;   // PART UNTI 02 DONE IN TRANSIT
            COOLING_DONE : Bool;   // PART COOLING DONE
            INSPECTION_DONE : Bool;   // PART INSPECTION DONE
            OUTFEED_CAMARA_OK : Bool;   // PART OUTFEED CAMARA OK
            SPARE2 : Bool;
            SPARE3 : Bool;
            SPARE4 : Bool;
            SPARE5 : Bool;
            SPARE6 : Bool;   // PART ROTATION 2 NEW PART
            SPARE7 : Bool;
            SPARE8 : Bool;
            SPARE9 : Bool;
            SPARE10 : Bool;
            SPARE11 : Bool;
            SPARE12 : Bool;
         END_STRUCT;
      END_STRUCT;
      PART_ID : Array[0..99] of Char;   // PART ID
      SPARE : Array[0..10] of Byte;
   END_STRUCT;
END_TYPE

TYPE "ABB_INPUTS"
// stored: IsFailsafeCompliant false
   STRUCT
      SYSTEM_SIGNAL : Struct
         SYS_STOP : Bool;   // MACHINE HEARTBEAT (MACHINE TO GANTRY) / STOP EXECUTION PROGRAM
         SYS_MOTOR_OFF : Bool;   // TURN OFF MOTORS
         SYS_RESET_E_STOP : Bool;   // MACHINE EMERGENCY STOP OK (MACHINE TO GANTRY) / RESET EMERGENCY STOP
         SYS_STOP_CYCLE : Bool;   // MACHINE SAFETY GATES OK (LOCKED)(MACHINE TO GANTRY) / STOP PROGRAM - END OF CYCLE
         SYS_RESET_ERROR : Bool;   // MACHINE IN MANUAL MODE (MACHINE TO GANTRY) / RESET EXECUTION ERROR
         SYS_START_MAIN : Bool;   // MACHINE IN AUTO MODE(MACHINE TO GANTRY) / START MAIN PROGRAM
         SYS_START : Bool;   // MACHINE AUTO CYCLE RUNNING (MACHINE TO GANTRY) / START PROGRAM(CONTINUE)
         SYS_MOTOR_ON : Bool;   // MACHINE IS IN WARMUP CYCLE (MACHINE TO GANTRY) / TURN ON MOTORS
         SPARE_65_0 : Byte;   // MACHINE IN RUN OUT MODE (MACHINE TO GANTRY)
         SPARE_66_0 : Byte;   // MACHINE PART DEMAND SOON (MACHINE TO GANTRY)
         SPARE_67_0 : Byte;
      END_STRUCT;
      GENERAL_SIGNAL : Struct
         STYLE_INIT : Bool;   // GANTRY HEARTBEAT (GANTRY TO MACHINE) / INITIATE STYLE
         READ_DEC_CODE : Bool;   // READ DECISION CODE
         OK_CONTINUE : Bool;   // GANTRY EMERGENCY STOP OK (GANTRY TO MACHINE) / OK TO CONTINUE
         ENTER_REQUEST : Bool;   // ENTER CELL REQUEST
         DRY_CYCLE : Bool;   // GANTRY IN MANUAL MODE (GANTRY TO MACHINE) / DRY CYCLE
         RECOVER_REQ : Bool;   // GANTRY IN AUTO MODE (GANTRY TO MACHINE) / RECOVERY REQUEST
         SPARE_68_6 : Bool;   // GANTRY IN AUTO CYCLE RUNNING (GANTRY TO MACHINE)
         SPARE_68_7 : Bool;   // GANTRY OVERHEAD DOOR CLOSED & LOCKED (GANTRY TO MACHINE)
         IMMEDIATE_STOP_AUX : Bool;
         STOP_END_OF_CYCLE : Bool;
         RUNOUT_REQUEST : Bool;
         SPARE_69_3 : Bool;
         SPARE_69_4 : Bool;
         SPARE_69_5 : Bool;
         SPARE_69_6 : Bool;
         SPARE_69_7 : Bool;
         SPARE_70_0 : Byte;   // GANTRY CLEAR OF MACHINE (GANTRY TO MACHINE)
         SPARE_71_0 : Byte;   // GANTRY CLEAR OF FIXTURE (GANTRY TO MACHINE)
         SPARE_72_0 : Byte;
         SPARE_73_0 : Byte;
      END_STRUCT;
      PROGRAM : Struct
         STYLE_PROGRAM : Byte;   // GANTRY HEARTBEAT (GANTRY TO MACHINE) / GROUP INPUT INDICATING STYLE NUMBER PROGRAM
         DEC_CODE : Byte;   // SPECIFIC OPERATING WITHIN A STYLE
         PART_TYPE : Byte;   // GANTRY EMERGENCY STOP OK (GANTRY TO MACHINE) / PART TYPE SELECTED
         SPARE_77_0 : Byte;   // GANTRY EMERGENCY STOP OK (GANTRY TO MACHINE)
      END_STRUCT;
      GRIPPERS : Struct
         T1_GRIPPER_A_OPEN_REQ : Bool;   // ROBOT TOOL 1 GRIPPER A OPEN REQUEST
         T1_GRIPPER_A_CLOSE_REQ : Bool;   // ROBOT TOOL 1 GRIPPER A CLOSE REQUEST
         SPARE_78_2 : Bool;
         SPARE_78_3 : Bool;
         T1_GRIPPER_A_OPEN : Bool;   // ROBOT TOOL 1 GRIPPER A OPEN
         T1_GRIPPER_A_CLOSED : Bool;   // ROBOT TOOL 1 GRIPPER A CLOSED
         SPARE_78_6 : Bool;
         SPARE_78_7 : Bool;
         T1_GRIPPER_B_OPEN_REQ : Bool;   // ROBOT TOOL 1 GRIPPER B OPEN REQUEST
         T1_GRIPPER_B_CLOSE_REQ : Bool;   // ROBOT TOOL 1 GRIPPER B CLOSE REQUEST
         SPARE_79_2 : Bool;
         SPARE_79_3 : Bool;
         T1_GRIPPER_B_OPEN : Bool;   // ROBOT TOOL 1 GRIPPER B OPEN
         T1_GRIPPER_B_CLOSED : Bool;   // ROBOT TOOL 1 GRIPPER B CLOSED
         SPARE_79_6 : Bool;
         SPARE_79_7 : Bool;
         T1_GRIPPER_C_OPEN_REQ : Bool;   // ROBOT TOOL 1 GRIPPER C OPEN REQUEST
         T1_GRIPPER_C_CLOSE_REQ : Bool;   // ROBOT TOOL 1 GRIPPER C CLOSE REQUEST
         SPARE_80_2 : Bool;
         SPARE_80_3 : Bool;
         T1_GRIPPER_C_OPEN : Bool;   // ROBOT TOOL 1 GRIPPER C OPEN
         T1_GRIPPER_C_CLOSED : Bool;   // ROBOT TOOL 1 GRIPPER C CLOSED
         SPARE_80_6 : Bool;
         SPARE_80_7 : Bool;
         T1_GRIPPER_D_OPEN_REQ : Bool;   // ROBOT TOOL 1 GRIPPER D OPEN REQUEST
         T1_GRIPPER_D_CLOSE_REQ : Bool;   // ROBOT TOOL 1 GRIPPER D CLOSE REQUEST
         SPARE_81_2 : Bool;
         SPARE_81_3 : Bool;
         T1_GRIPPER_D_OPEN : Bool;   // ROBOT TOOL 1 GRIPPER D OPEN
         T1_GRIPPER_D_CLOSED : Bool;   // ROBOT TOOL 1 GRIPPER D CLOSED
         SPARE_81_6 : Bool;
         SPARE_81_7 : Bool;
         T1_GRIPPER_E_OPEN_REQ : Bool;   // ROBOT TOOL 1 GRIPPER E OPEN REQUEST
         T1_GRIPPER_E_CLOSE_REQ : Bool;   // ROBOT TOOL 1 GRIPPER E CLOSE REQUEST
         SPARE_82_2 : Bool;
         SPARE_82_3 : Bool;
         T1_GRIPPER_E_OPEN : Bool;   // ROBOT TOOL 1 GRIPPER E OPEN
         T1_GRIPPER_E_CLOSED : Bool;   // ROBOT TOOL 1 GRIPPER E CLOSED
         SPARE_82_6 : Bool;
         SPARE_82_7 : Bool;
         T2_GRIPPER_A_OPEN_REQ : Bool;   // ROBOT TOOL 2 GRIPPER A OPEN REQUEST
         T2_GRIPPER_A_CLOSE_REQ : Bool;   // ROBOT TOOL 2 GRIPPER A CLOSE REQUEST
         SPARE_83_2 : Bool;
         SPARE_83_3 : Bool;
         T2_GRIPPER_A_OPEN : Bool;   // ROBOT TOOL 2 GRIPPER A OPEN
         T2_GRIPPER_A_CLOSED : Bool;   // ROBOT TOOL 2 GRIPPER A CLOSED
         SPARE_83_6 : Bool;
         SPARE_83_7 : Bool;
         T2_GRIPPER_B_OPEN_REQ : Bool;   // ROBOT TOOL 2 GRIPPER B OPEN REQUEST
         T2_GRIPPER_B_CLOSE_REQ : Bool;   // ROBOT TOOL 2 GRIPPER B CLOSE REQUEST
         SPARE_84_2 : Bool;
         SPARE_84_3 : Bool;
         T2_GRIPPER_B_OPEN : Bool;   // ROBOT TOOL 2 GRIPPER B OPEN
         T2_GRIPPER_B_CLOSED : Bool;   // ROBOT TOOL 2 GRIPPER B CLOSED
         SPARE_84_6 : Bool;
         SPARE_84_7 : Bool;
         T2_GRIPPER_C_OPEN_REQ : Bool;   // ROBOT TOOL 2 GRIPPER C OPEN REQUEST
         T2_GRIPPER_C_CLOSE_REQ : Bool;   // ROBOT TOOL 2 GRIPPER C CLOSE REQUEST
         SPARE_85_2 : Bool;
         SPARE_85_3 : Bool;
         T2_GRIPPER_C_OPEN : Bool;   // ROBOT TOOL 2 GRIPPER C OPEN
         T2_GRIPPER_C_CLOSED : Bool;   // ROBOT TOOL 2 GRIPPER C CLOSED
         SPARE_85_6 : Bool;
         SPARE_85_7 : Bool;
         T2_GRIPPER_D_OPEN_REQ : Bool;   // ROBOT TOOL 2 GRIPPER D OPEN REQUEST
         T2_GRIPPER_D_CLOSE_REQ : Bool;   // ROBOT TOOL 2 GRIPPER D CLOSE REQUEST
         SPARE_86_2 : Bool;
         SPARE_86_3 : Bool;
         T2_GRIPPER_D_OPEN : Bool;   // ROBOT TOOL 2 GRIPPER D OPEN
         T2_GRIPPER_D_CLOSED : Bool;   // ROBOT TOOL 2 GRIPPER D CLOSED
         SPARE_86_6 : Bool;
         SPARE_86_7 : Bool;
         T2_GRIPPER_E_OPEN_REQ : Bool;   // ROBOT TOOL 2 GRIPPER E OPEN REQUEST
         T2_GRIPPER_E_CLOSE_REQ : Bool;   // ROBOT TOOL 2 GRIPPER E CLOSE REQUEST
         SPARE_87_2 : Bool;
         SPARE_87_3 : Bool;
         T2_GRIPPER_E_OPEN : Bool;   // ROBOT TOOL 2 GRIPPER E OPEN
         T2_GRIPPER_E_CLOSED : Bool;   // ROBOT TOOL 2 GRIPPER E CLOSED
         SPARE_87_6 : Bool;
         SPARE_87_7 : Bool;
         T1_ALL_GRIPS_OPEN_REQ : Bool;   // ROBOT TOOL 1 OPEN ALL GRIPPERS REQUEST
         T1_ALL_GRIPS_CLOSE_REQ : Bool;   // ROBOT TOOL 1 CLOSE ALL GRIPPERS REQUEST
         T1_ALL_GRIPPERS_OPEN : Bool;   // ROBOT TOOL 1 ALL GRIPPERS OPEN
         T1_ALL_GRIPPERS_CLOSED : Bool;   // ROBOT TOOL 1 ALL GRIPPERS CLOSED
         SPARE_88_4 : Bool;
         SPARE_88_5 : Bool;
         SPARE_88_6 : Bool;
         SPARE_88_7 : Bool;
         T2_ALL_GRIPS_OPEN_REQ : Bool;   // ROBOT TOOL 2 CLOSE ALL GRIPPERS REQUEST
         T2_ALL_GRIPS_CLOSE_REQ : Bool;   // ROBOT TOOL 2 CLOSE ALL GRIPPERS REQUEST
         T2_ALL_GRIPPERS_OPEN : Bool;   // ROBOT TOOL 2 ALL GRIPPERS OPEN
         T2_ALL_GRIPPERS_CLOSED : Bool;   // ROBOT TOOL 2 ALL GRIPPERS CLOSED
         SPARE_89_4 : Bool;
         SPARE_89_5 : Bool;
         SPARE_89_6 : Bool;
         SPARE_89_7 : Bool;
         SPARE_90_0 : Byte;
         FAULT_NUMBER : Byte;   // FAULT RESPONSE
      END_STRUCT;
      CLEARS : Struct
         CLEAR_U_1 : Bool;   // GANTRY HEARTBEAT (GANTRY TO MACHINE) / CLEAR TO GET IN UNIT 1
         CLEAR_U_2 : Bool;   // CLEAR TO GET IN UNIT 2
         CLEAR_U_3 : Bool;   // GANTRY EMERGENCY STOP OK (GANTRY TO MACHINE) / CLEAR TO GET IN UNIT 3
         CLEAR_U_4 : Bool;   // CLEAR TO GET IN UNIT 4
         CLEAR_U_5 : Bool;   // GANTRY IN MANUAL MODE (GANTRY TO MACHINE) / CLEAR TO GET IN UNIT 5
         CLEAR_U_6 : Bool;   // GANTRY IN AUTO MODE (GANTRY TO MACHINE) / CLEAR TO GET IN UNIT 6
         CLEAR_U_7 : Bool;   // GANTRY IN AUTO CYCLE RUNNING (GANTRY TO MACHINE) / CLEAR TO GET IN UNIT 7
         CLEAR_U_8 : Bool;   // GANTRY OVERHEAD DOOR CLOSED & LOCKED (GANTRY TO MACHINE) / CLEAR TO GET IN UNIT 8
         CLEAR_U_9 : Bool;   // GANTRY IN RUN OUT COMPLETE(GANTRY TO MACHINE) / CLEAR TO GET IN UNIT 9
         CLEAR_U_10 : Bool;   // GANTRY CLEAR OF MACHINE (GANTRY TO MACHINE) / CLEAR TO GET IN UNIT 10
         SPARE_93_2 : Bool;   // GANTRY CLEAR OF FIXTURE (GANTRY TO MACHINE)
         SPARE_93_3 : Bool;
         SPARE_93_4 : Bool;
         SPARE_93_5 : Bool;   // GANTRY PART TYPE CHANGE REQUESTED (GANTRY TO MACHINE)
         SPARE_93_6 : Bool;   // GANTRY REQUEST MACHINE TO RUN WITH LOADED PARTS (GANTRY TO MACHINE)
         SPARE_93_7 : Bool;   // GANTRY RUN OUT REQUESTED (GANTRY TO MACHINE)
         SPARE_94_0 : Byte;
         SPARE_95_0 : Byte;
      END_STRUCT;
      TASKS : Struct
         COMPLETE_TSK_1 : Bool;   // GANTRY HEARTBEAT (GANTRY TO MACHINE) / PICK REQUEST - ST1
         COMPLETE_TSK_2 : Bool;   // PLACE REQUEST - ST1
         COMPLETE_TSK_3 : Bool;   // GANTRY EMERGENCY STOP OK (GANTRY TO MACHINE) / PICK&PLACE REQUEST - ST1
         COMPLETE_TSK_4 : Bool;   // ROBOT COMPLETE TASK 4
         COMPLETE_TSK_5 : Bool;   // GANTRY IN MANUAL MODE (GANTRY TO MACHINE) / ROBOT COMPLETE TASK 5
         COMPLETE_TSK_6 : Bool;   // GANTRY IN AUTO MODE (GANTRY TO MACHINE) / ROBOT COMPLETE TASK 6
         COMPLETE_TSK_7 : Bool;   // GANTRY IN AUTO CYCLE RUNNING (GANTRY TO MACHINE) / ROBOT COMPLETE TASK 7
         COMPLETE_TSK_8 : Bool;   // GANTRY OVERHEAD DOOR CLOSED & LOCKED (GANTRY TO MACHINE) / ROBOT COMPLETE TASK 8
         SPARE_97_0 : Byte;   // GANTRY IN RUN OUT COMPLETE(GANTRY TO MACHINE)
         SPARE_98_0 : Byte;   // GANTRY CLEAR OF MACHINE (GANTRY TO MACHINE)
         SPARE_99_0 : Byte;   // GANTRY CLEAR OF FIXTURE (GANTRY TO MACHINE)
         SPARE_100_0 : Byte;
         SPARE_101_0 : Byte;
         SPARE_102_0 : Byte;
         SPARE_103_0 : Byte;
      END_STRUCT;
      PARTS_ENABLED : Struct
         PART_A_ENABLED : Bool;   // GANTRY HEARTBEAT (GANTRY TO MACHINE) / PART A ENABLED TO WORK
         PART_B_ENABLED : Bool;   // PART B ENABLED TO WORK
         PART_C_ENABLED : Bool;   // GANTRY EMERGENCY STOP OK (GANTRY TO MACHINE) / PART C ENABLED TO WORK
         PART_D_ENABLED : Bool;   // PART D ENABLED TO WORK
         PART_E_ENABLED : Bool;   // GANTRY IN MANUAL MODE (GANTRY TO MACHINE) / PART E ENABLED TO WORK
         SPARE_104_5 : Bool;   // GANTRY IN AUTO MODE (GANTRY TO MACHINE)
         SPARE_104_6 : Bool;   // GANTRY IN AUTO CYCLE RUNNING (GANTRY TO MACHINE)
         SPARE_104_7 : Bool;   // GANTRY OVERHEAD DOOR CLOSED & LOCKED (GANTRY TO MACHINE)
         SPARE_105_0 : Byte;   // GANTRY CLEAR OF FIXTURE (GANTRY TO MACHINE)
      END_STRUCT;
      SPARES : Array[106..127] of Byte;
   END_STRUCT;
END_TYPE

TYPE "ABB_OUTPUTS"
// stored: IsFailsafeCompliant false
   STRUCT
      SYSTEM_SIGNAL : Struct
         SYS_MOTOR_ON : Bool;   // MACHINE HEARTBEAT (MACHINE TO GANTRY) / MOTORS ON STATE
         SYS_MOTOR_OFF : Bool;   // MOTORS OFF STATE
         SYS_CYCLE_ON : Bool;   // MACHINE EMERGENCY STOP OK (MACHINE TO GANTRY) / ROBOT IN CYCLE ON STATE
         SYS_AUTO_ON : Bool;   // MACHINE SAFETY GATES OK (LOCKED)(MACHINE TO GANTRY) / ROBOT IN AUTO MODE
         SYS_EMERG_UOP : Bool;   // MACHINE IN MANUAL MODE (MACHINE TO GANTRY) / EMERGENCY STOP ACTIVE
         SYS_ERROR : Bool;   // MACHINE IN AUTO MODE(MACHINE TO GANTRY) / EXECUTION ERROR ACTIVE
         SPARE_0_6 : Bool;   // MACHINE AUTO CYCLE RUNNING (MACHINE TO GANTRY)
         SPARE_0_7 : Bool;   // MACHINE IS IN WARMUP CYCLE (MACHINE TO GANTRY)
         SPARE_1_0 : Byte;   // MACHINE IN RUN OUT MODE (MACHINE TO GANTRY)
         SPARE_2_0 : Byte;   // MACHINE PART DEMAND SOON (MACHINE TO GANTRY)
         SPARE_3_0 : Byte;
      END_STRUCT;
      GENERAL_SIGNAL : Struct
         STYLE_INIT_ACK : Bool;   // GANTRY HEARTBEAT (GANTRY TO MACHINE) / ACKNOWLEDGE INITIATE STYLE
         IN_CYCLE : Bool;   // IN CYCLE
         REQ_TO_CONT : Bool;   // GANTRY EMERGENCY STOP OK (GANTRY TO MACHINE) / REQUEST TO CONTINUE
         DRY_CYCLE : Bool;   // DRY CYCLE MODE
         RBT_100_SPD : Bool;   // GANTRY IN MANUAL MODE (GANTRY TO MACHINE) / ROBOT 100% SPEED
         RBT_HEARTBEAT : Bool;   // GANTRY IN AUTO MODE (GANTRY TO MACHINE) / ROBOT HEARTBEAT SIGNAL
         "OP_PANEL_E-STOP" : Bool;   // GANTRY IN AUTO CYCLE RUNNING (GANTRY TO MACHINE) / OPERATOR PANEL E-STOP
         "TEACH_PENDANT_E-STOP" : Bool;   // GANTRY OVERHEAD DOOR CLOSED & LOCKED (GANTRY TO MACHINE) / TEACH PENDANT E-STOP
         EXT_ENABLED : Bool;   // GANTRY IN RUN OUT COMPLETE(GANTRY TO MACHINE) / EXTERNAL E-STOP
         DEAD_ENABLED : Bool;   // GANTRY CLEAR OF MACHINE (GANTRY TO MACHINE) / DEADMAN E-STOP
         "I/O_SIMULATE" : Bool;   // GANTRY CLEAR OF FIXTURE (GANTRY TO MACHINE) / I/O SIMULATED
         SRV_DISC_OFF : Bool;   // SERVO DISABLED OFF
         SRV_BATT_ALARM : Bool;   // LOW BATTERY ALARM ON SERVO
         TASK_OK : Bool;   // TASK OK
         STEP_MODE_ON : Bool;   // STEP MODE STATUS
         AUTO_MODE_ON : Bool;   // SELECTOR SWITCH IS SET TO AUTO
         MANUAL_ON : Bool;   // SELECTOR SWITCH IS SET TO MANUAL
         FENCE_OPEN : Bool;   // FENCE IS OPEN
         INTERLOCK : Bool;   // ROBOT IN INTERLOCK
         ROUT_ACTIVE : Bool;   // ROUTER ACTIVE BIT
         FAULT_RSP_ACK : Bool;   // HMI OPTION FAULT RESPONSE
         DCS_SIGN_MATCH : Bool;   // DCS SIGNATURE MATCH
         REQ_DEC_CODE : Bool;   // REQUEST DECITION
         FLT_TASK_UOPPED : Bool;   // ROBOT TASK STOPPED
         FLT_COLLISION : Bool;   // ROBOT COLLITION FAULT
         FLT_BAD_PLC_INPUT : Bool;   // BAD PLC INPUT
         FLT_GRIP_LOW_PRS : Bool;   // ROBOT GRIPPER PRESSURE LOW
         FLT_BAD_OPTN : Bool;   // BAD PLC FAULT RESPONSE
         RECOV_AT_MAIN : Bool;   // RECOVERY POINTER TO MAIN
         FLT_USER_BIT_8 : Bool;   // USER DEFINABLE FAULT BIT
         SPARE_7_6 : Bool;
         SPARE_7_7 : Bool;
         SPARE_8_0 : Byte;
         SPARE_9_0 : Byte;
      END_STRUCT;
      PROGRAM : Struct
         STYLE_PROGRAM_ACK : Byte;   // GANTRY HEARTBEAT (GANTRY TO MACHINE) / SELECT STYLE PROGRAM ACKNOWLEDGE
         DEC_CODE_ACK : Byte;   // SELECT DECITION CODE ACKNOWLEDGE
         PART_TYPE_ACK : Byte;   // GANTRY EMERGENCY STOP OK (GANTRY TO MACHINE) / PART TYPE ACKNOWLEDGE
         SPARE_13_0 : Byte;   // GANTRY EMERGENCY STOP OK (GANTRY TO MACHINE)
      END_STRUCT;
      GRIPPERS : Struct
         T1_GRIPPER_A_OPEN_REQ : Bool;   // ROBOT TOOL 1 GRIPPER A OPEN REQUEST
         T1_GRIPPER_A_CLOSE_REQ : Bool;   // ROBOT TOOL 1 GRIPPER A CLOSE REQUEST
         SPARE_14_2 : Bool;
         SPARE_14_3 : Bool;
         T1_GRIPPER_A_OPEN : Bool;   // ROBOT TOOL 1 GRIPPER A OPEN
         T1_GRIPPER_A_CLOSED : Bool;   // ROBOT TOOL 1 GRIPPER A CLOSED
         SPARE_14_6 : Bool;
         SPARE_14_7 : Bool;
         T1_GRIPPER_B_OPEN_REQ : Bool;   // ROBOT TOOL 1 GRIPPER B OPEN REQUEST
         T1_GRIPPER_B_CLOSE_REQ : Bool;   // ROBOT TOOL 1 GRIPPER B CLOSE REQUEST
         SPARE_15_2 : Bool;
         SPARE_15_3 : Bool;
         T1_GRIPPER_B_OPEN : Bool;   // ROBOT TOOL 1 GRIPPER B OPEN
         T1_GRIPPER_B_CLOSED : Bool;   // ROBOT TOOL 1 GRIPPER B CLOSED
         SPARE_15_6 : Bool;
         SPARE_15_7 : Bool;
         T1_GRIPPER_C_OPEN_REQ : Bool;   // ROBOT TOOL 1 GRIPPER C OPEN REQUEST
         T1_GRIPPER_C_CLOSE_REQ : Bool;   // ROBOT TOOL 1 GRIPPER C CLOSE REQUEST
         SPARE_16_2 : Bool;
         SPARE_16_3 : Bool;
         T1_GRIPPER_C_OPEN : Bool;   // ROBOT TOOL 1 GRIPPER C OPEN
         T1_GRIPPER_C_CLOSED : Bool;   // ROBOT TOOL 1 GRIPPER C CLOSED
         SPARE_16_6 : Bool;
         SPARE_16_7 : Bool;
         T1_GRIPPER_D_OPEN_REQ : Bool;   // ROBOT TOOL 1 GRIPPER D OPEN REQUEST
         T1_GRIPPER_D_CLOSE_REQ : Bool;   // ROBOT TOOL 1 GRIPPER D CLOSE REQUEST
         SPARE_17_2 : Bool;
         SPARE_17_3 : Bool;
         T1_GRIPPER_D_OPEN : Bool;   // ROBOT TOOL 1 GRIPPER D OPEN
         T1_GRIPPER_D_CLOSED : Bool;   // ROBOT TOOL 1 GRIPPER D CLOSED
         SPARE_17_6 : Bool;
         SPARE_17_7 : Bool;
         T1_GRIPPER_E_OPEN_REQ : Bool;   // ROBOT TOOL 1 GRIPPER E OPEN REQUEST
         T1_GRIPPER_E_CLOSE_REQ : Bool;   // ROBOT TOOL 1 GRIPPER E CLOSE REQUEST
         SPARE_18_2 : Bool;
         SPARE_18_3 : Bool;
         T1_GRIPPER_E_OPEN : Bool;   // ROBOT TOOL 1 GRIPPER E OPEN
         T1_GRIPPER_E_CLOSED : Bool;   // ROBOT TOOL 1 GRIPPER E CLOSED
         SPARE_18_6 : Bool;
         SPARE_18_7 : Bool;
         T2_GRIPPER_A_OPEN_REQ : Bool;   // ROBOT TOOL 2 GRIPPER A OPEN REQUEST
         T2_GRIPPER_A_CLOSE_REQ : Bool;   // ROBOT TOOL 2 GRIPPER A CLOSE REQUEST
         SPARE_19_2 : Bool;
         SPARE_19_3 : Bool;
         T2_GRIPPER_A_OPEN : Bool;   // ROBOT TOOL 2 GRIPPER A OPEN
         T2_GRIPPER_A_CLOSED : Bool;   // ROBOT TOOL 2 GRIPPER A CLOSED
         SPARE_19_6 : Bool;
         SPARE_19_7 : Bool;
         T2_GRIPPER_B_OPEN_REQ : Bool;   // ROBOT TOOL 2 GRIPPER B OPEN REQUEST
         T2_GRIPPER_B_CLOSE_REQ : Bool;   // ROBOT TOOL 2 GRIPPER B CLOSE REQUEST
         SPARE_20_2 : Bool;
         SPARE_20_3 : Bool;
         T2_GRIPPER_B_OPEN : Bool;   // ROBOT TOOL 2 GRIPPER B OPEN
         T2_GRIPPER_B_CLOSED : Bool;   // ROBOT TOOL 2 GRIPPER B CLOSED
         SPARE_20_6 : Bool;
         SPARE_20_7 : Bool;
         T2_GRIPPER_C_OPEN_REQ : Bool;   // ROBOT TOOL 2 GRIPPER C OPEN REQUEST
         T2_GRIPPER_C_CLOSE_REQ : Bool;   // ROBOT TOOL 2 GRIPPER C CLOSE REQUEST
         SPARE_21_2 : Bool;
         SPARE_21_3 : Bool;
         T2_GRIPPER_C_OPEN : Bool;   // ROBOT TOOL 2 GRIPPER C OPEN
         T2_GRIPPER_C_CLOSED : Bool;   // ROBOT TOOL 2 GRIPPER C CLOSED
         SPARE_21_6 : Bool;
         SPARE_21_7 : Bool;
         T2_GRIPPER_D_OPEN_REQ : Bool;   // ROBOT TOOL 2 GRIPPER D OPEN REQUEST
         T2_GRIPPER_D_CLOSE_REQ : Bool;   // ROBOT TOOL 2 GRIPPER D CLOSE REQUEST
         SPARE_22_2 : Bool;
         SPARE_22_3 : Bool;
         T2_GRIPPER_D_OPEN : Bool;   // ROBOT TOOL 2 GRIPPER D OPEN
         T2_GRIPPER_D_CLOSED : Bool;   // ROBOT TOOL 2 GRIPPER D CLOSED
         SPARE_22_6 : Bool;
         SPARE_22_7 : Bool;
         T2_GRIPPER_E_OPEN_REQ : Bool;   // ROBOT TOOL 2 GRIPPER E OPEN REQUEST
         T2_GRIPPER_E_CLOSE_REQ : Bool;   // ROBOT TOOL 2 GRIPPER E CLOSE REQUEST
         SPARE_23_2 : Bool;
         SPARE_23_3 : Bool;
         T2_GRIPPER_E_OPEN : Bool;   // ROBOT TOOL 2 GRIPPER E OPEN
         T2_GRIPPER_E_CLOSED : Bool;   // ROBOT TOOL 2 GRIPPER E CLOSED
         SPARE_23_6 : Bool;
         SPARE_23_7 : Bool;
         T1_ALL_GRIPS_OPEN_REQ : Bool;   // ROBOT TOOL 1 OPEN ALL GRIPPERS REQUEST
         T1_ALL_GRIPS_CLOSE_REQ : Bool;   // ROBOT TOOL 1 CLOSE ALL GRIPPERS REQUEST
         T1_ALL_GRIPPERS_OPEN : Bool;   // ROBOT TOOL 1 ALL GRIPPERS OPEN
         T1_ALL_GRIPPERS_CLOSED : Bool;   // ROBOT TOOL 1 ALL GRIPPERS CLOSED
         SPARE_24_4 : Bool;
         SPARE_24_5 : Bool;
         SPARE_24_6 : Bool;
         SPARE_24_7 : Bool;
         T2_ALL_GRIPS_OPEN_REQ : Bool;   // ROBOT TOOL 2 CLOSE ALL GRIPPERS REQUEST
         T2_ALL_GRIPS_CLOSE_REQ : Bool;   // ROBOT TOOL 2 CLOSE ALL GRIPPERS REQUEST
         T2_ALL_GRIPPERS_OPEN : Bool;   // ROBOT TOOL 2 ALL GRIPPERS OPEN
         T2_ALL_GRIPPERS_CLOSED : Bool;   // ROBOT TOOL 2 ALL GRIPPERS CLOSED
         SPARE_25_4 : Bool;
         SPARE_25_5 : Bool;
         SPARE_25_6 : Bool;
         SPARE_25_7 : Bool;
         SPARE_26_0 : Byte;
         FAULT_NUMBER : Byte;   // FAULT RESPONSE
      END_STRUCT;
      CLEARS : Struct
         CLEAR_U_1_ACK : Bool;   // GANTRY HEARTBEAT (GANTRY TO MACHINE) / CLEAR UNIT 1
         CLEAR_U_2_ACK : Bool;   // CLEAR UNIT 2
         CLEAR_U_3_ACK : Bool;   // GANTRY EMERGENCY STOP OK (GANTRY TO MACHINE) / CLEAR UNIT 3
         CLEAR_U_4_ACK : Bool;   // CLEAR UNIT 4
         CLEAR_U_5_ACK : Bool;   // GANTRY IN MANUAL MODE (GANTRY TO MACHINE) / CLEAR UNIT 5
         CLEAR_U_6_ACK : Bool;   // GANTRY IN AUTO MODE (GANTRY TO MACHINE) / CLEAR UNIT 6
         CLEAR_U_7_ACK : Bool;   // GANTRY IN AUTO CYCLE RUNNING (GANTRY TO MACHINE) / CLEAR UNIT 7
         CLEAR_U_8_ACK : Bool;   // GANTRY OVERHEAD DOOR CLOSED & LOCKED (GANTRY TO MACHINE) / CLEAR UNIT 8
         CLEAR_U_9_ACK : Bool;   // GANTRY IN RUN OUT COMPLETE(GANTRY TO MACHINE) / CLEAR UNIT 9
         CLEAR_U_10_ACK : Bool;   // GANTRY CLEAR OF MACHINE (GANTRY TO MACHINE) / CLEAR UNIT 10
         SPARE_29_2 : Bool;   // GANTRY CLEAR OF FIXTURE (GANTRY TO MACHINE)
         SPARE_29_3 : Bool;
         SPARE_29_4 : Bool;
         SPARE_29_5 : Bool;   // GANTRY PART TYPE CHANGE REQUESTED (GANTRY TO MACHINE)
         SPARE_29_6 : Bool;   // GANTRY REQUEST MACHINE TO RUN WITH LOADED PARTS (GANTRY TO MACHINE)
         SPARE_29_7 : Bool;   // GANTRY RUN OUT REQUESTED (GANTRY TO MACHINE)
         SPARE_30_0 : Byte;
         SPARE_31_0 : Byte;
      END_STRUCT;
      TASKS : Struct
         TSK_COMPLETED_1 : Bool;   // GANTRY HEARTBEAT (GANTRY TO MACHINE) / ROBOT TASK 1 COMPLETED
         TSK_COMPLETED_2 : Bool;   // ROBOT TASK 2 COMPLETED
         TSK_COMPLETED_3 : Bool;   // GANTRY EMERGENCY STOP OK (GANTRY TO MACHINE) / ROBOT TASK 3 COMPLETED
         TSK_COMPLETED_4 : Bool;   // ROBOT TASK 4 COMPLETED
         TSK_COMPLETED_5 : Bool;   // GANTRY IN MANUAL MODE (GANTRY TO MACHINE) / ROBOT TASK 5 COMPLETED
         TSK_COMPLETED_6 : Bool;   // GANTRY IN AUTO MODE (GANTRY TO MACHINE) / ROBOT TASK 6 COMPLETED
         TSK_COMPLETED_7 : Bool;   // GANTRY IN AUTO CYCLE RUNNING (GANTRY TO MACHINE) / ROBOT TASK 7 COMPLETED
         TSK_COMPLETED_8 : Bool;   // GANTRY OVERHEAD DOOR CLOSED & LOCKED (GANTRY TO MACHINE) / ROBOT TASK 8 COMPLETED
         SPARE_33_0 : Byte;   // GANTRY IN RUN OUT COMPLETE(GANTRY TO MACHINE) / ROBOT TASK 9 COMPLETED
         SPARE_34_0 : Byte;   // GANTRY CLEAR OF MACHINE (GANTRY TO MACHINE) / ROBOT TASK 10 COMPLETED
         SPARE_35_0 : Byte;   // GANTRY CLEAR OF FIXTURE (GANTRY TO MACHINE)
         SPARE_36_0 : Byte;
         SPARE_37_0 : Byte;
         SPARE_38_0 : Byte;
         SPARE_39_0 : Byte;
      END_STRUCT;
      POSITIONS : Struct
         HOME : Bool;   // GANTRY HEARTBEAT (GANTRY TO MACHINE) / ROBOT AT HOME POSITION
         MAINT : Bool;   // ROBOT AT MAINTENANCE POSITION
         REPAIR : Bool;   // GANTRY EMERGENCY STOP OK (GANTRY TO MACHINE) / ROBOT AT REPAIRED POSITION
         ALIGN : Bool;   // ROBOT AT ALIGNED POSITION
         SHIP : Bool;   // GANTRY IN MANUAL MODE (GANTRY TO MACHINE) / ROBOT AT SHIPPED POSITION
         SPARE_38_5 : Bool;   // GANTRY IN AUTO MODE (GANTRY TO MACHINE)
         SPARE_38_6 : Bool;   // GANTRY IN AUTO CYCLE RUNNING (GANTRY TO MACHINE)
         SPARE_38_7 : Bool;   // GANTRY OVERHEAD DOOR CLOSED & LOCKED (GANTRY TO MACHINE)
         UNIT_1 : Bool;   // GANTRY OVERHEAD DOOR CLOSED & LOCKED (GANTRY TO MACHINE) / ROBOT AT POUNCE POSITION UNIT 1
         UNIT_2 : Bool;   // GANTRY OVERHEAD DOOR CLOSED & LOCKED (GANTRY TO MACHINE) / ROBOT AT POUNCE POSITION UNIT 2
         UNIT_3 : Bool;   // GANTRY OVERHEAD DOOR CLOSED & LOCKED (GANTRY TO MACHINE) / ROBOT AT POUNCE POSITION UNIT 3
         UNIT_4 : Bool;   // GANTRY OVERHEAD DOOR CLOSED & LOCKED (GANTRY TO MACHINE) / ROBOT AT POUNCE POSITION UNIT 4
         UNIT_5 : Bool;   // GANTRY OVERHEAD DOOR CLOSED & LOCKED (GANTRY TO MACHINE) / ROBOT AT POUNCE POSITION UNIT 5
         UNIT_6 : Bool;   // GANTRY IN RUN OUT COMPLETE(GANTRY TO MACHINE) / ROBOT AT POUNCE POSITION UNIT 6
         UNIT_7 : Bool;   // GANTRY IN RUN OUT COMPLETE(GANTRY TO MACHINE) / ROBOT AT POUNCE POSITION UNIT 7
         UNIT_8 : Bool;   // GANTRY IN RUN OUT COMPLETE(GANTRY TO MACHINE) / ROBOT AT POUNCE POSITION UNIT 8
         SPARE_42_0 : Byte;   // GANTRY CLEAR OF MACHINE (GANTRY TO MACHINE)
         SPARE_43_0 : Byte;   // GANTRY CLEAR OF FIXTURE (GANTRY TO MACHINE)
         SPARE_44_0 : Byte;
         SPARE_45_0 : Byte;
      END_STRUCT;
      SPARES : Array[46..63] of Byte;
   END_STRUCT;
END_TYPE

TYPE "CELL_SEQUENCES"
// stored: IsFailsafeCompliant false
   STRUCT
      GENERAL_CONDITIONS : Bool;   // GENERAL CONDITIONS
      INITIAL_CONDITIONS : Bool;   // INITIAL CONDITIONS
      START_REQUEST : Bool;   // START REQUEST
      START_COMMAND : Bool;   // START COMMAND
      SPARE_0_4 : Bool;   // SPARE 0 4
      COMMAND_PULSE : Bool;   // COMMAND PULSE
      REQUEST_PULSE : Bool;   // REQUEST PULSE
      SEQUENCE_RUNNING : Bool;   // SEQUENCE RUNNING
      STEP_1 : Bool;   // STEP 1
      STEP_2 : Bool;   // STEP 2
      STEP_3 : Bool;   // STEP 3
      STEP_4 : Bool;   // STEP 4
      STEP_5 : Bool;   // STEP 5
      STEP_6 : Bool;   // STEP 6
      STEP_7 : Bool;   // STEP 7
      STEP_8 : Bool;   // STEP 8
      STEP_9 : Bool;   // STEP 9
      STEP_10 : Bool;   // STEP 10
      STEP_11 : Bool;   // STEP 11
      STEP_12 : Bool;   // STEP 12
      STEP_13 : Bool;   // STEP 13
      STEP_14 : Bool;   // STEP 14
      STEP_15 : Bool;   // STEP 15
      STEP_16 : Bool;   // STEP 16
      SPARE_3_0 : Byte;   // SPARE 3 0
      SPARE_4_0 : Byte;   // SPARE 4 0
      RESET_PLC_CNC : Bool;   // RESET PLC CNC
      SEMI_REQ : Bool;   // SEMI REQUEST
      AUTO_REQ : Bool;   // AUTO REQUEST
      TEACH_PENDANT_REQUEST : Bool;   // TEACH PENDANT REQUEST
      SPARE_5_4 : Bool;   // SPARE 5 4
      SPARE_5_5 : Bool;   // SPARE 5 5
      SPARE_5_6 : Bool;   // SPARE 5 6
      SEQ_DONE : Bool;   // SEQ DONE
      TIME_EXCEEDED : Bool;   // TIME EXCEEDED
      SPARE_6_1 : Bool;   // SPARE 6 1
      SPARE_6_2 : Bool;   // SPARE 6 2
      SPARE_6_3 : Bool;   // SPARE 6 3
      SPARE_6_4 : Bool;   // SPARE 6 4
      SPARE_6_5 : Bool;   // SPARE 6 5
      SPARE_6_6 : Bool;   // SPARE 6 6
      SPARE_6_7 : Bool;   // SPARE 6 7
      WARNING : Bool;   // WARNING
      HELP : Bool;   // HELP
      SPARE_7_2 : Bool;   // SPARE 7 2
      SPARE_7_3 : Bool;   // SPARE 7 3
      SPARE_7_4 : Bool;   // SPARE 7 4
      SPARE_7_5 : Bool;   // SPARE 7 5
      SPARE_7_6 : Bool;   // SPARE 7 6
      SPARE_7_7 : Bool;   // SPARE 7 7
      AUX0 : Bool;   // AUX0
      AUX1 : Bool;   // AUX1
      AUX2 : Bool;   // AUX2
      AUX3 : Bool;   // AUX3
      WARNING_GONE : Bool;   // WARNING GONE
      AUX5 : Bool;   // AUX5
      AUX6 : Bool;   // AUX6
      AUX7 : Bool;   // AUX7
      START_GRAL_COND_HELP : Bool;   // START GENERAL COND HELP
      START_INIT_COND_HELP : Bool;   // START INITIAL COND HELP
      STOP_GRAL_HELP : Bool;   // STOP GENERAL HELP
      STOP_INIT_HELP : Bool;   // STOP INITIAL HELP
      SPARE_9_4 : Bool;   // SPARE 9 4
      SPARE_9_5 : Bool;   // SPARE 9 5
      GRAL_COND_HELP : Bool;   // GENERAL COND HELP
      INIT_COND_HELP : Bool;   // INITIAL COND HELP
      SPARE_10_0 : Byte;
      "TIMER_TIME _EXCEED" : TON_TIME;   // CELL SEQUENCE TIMER TIME EXCEEDED
   END_STRUCT;
   // "TIMER_TIME _EXCEED".PT := T#20S;
END_TYPE

TYPE "FANUC_INPUTS"
// stored: IsFailsafeCompliant false
   STRUCT
      SYSTEM_SIGNAL : Struct
         SYS_IMSTP : Bool;   // MACHINE HEARTBEAT (MACHINE TO GANTRY) / IMMEDIATE STOP
         SYS_HOLD : Bool;   // HOLD ROBOT
         SYS_SFSPD : Bool;   // MACHINE EMERGENCY STOP OK (MACHINE TO GANTRY) / SAFE SPEED
         SYS_CYCLE_STOP : Bool;   // MACHINE SAFETY GATES OK (LOCKED)(MACHINE TO GANTRY) / CYCLE STOP
         SYS_FAULT_RESET : Bool;   // MACHINE IN MANUAL MODE (MACHINE TO GANTRY) / FAULT RESET
         SYS_HOME : Bool;   // MACHINE IN AUTO MODE(MACHINE TO GANTRY) / HOME
         SYS_START : Bool;   // MACHINE AUTO CYCLE RUNNING (MACHINE TO GANTRY) / START PROGRAM / CONTINUE PROGRAM
         SYS_MOTION_ENBL : Bool;   // MACHINE IS IN WARMUP CYCLE (MACHINE TO GANTRY) / MOTION ENABLE
         SPARE_65_0 : Byte;   // MACHINE IN RUN OUT MODE (MACHINE TO GANTRY)
         SPARE_66_0 : Byte;   // MACHINE PART DEMAND SOON (MACHINE TO GANTRY)
         SPARE_67_0 : Byte;
      END_STRUCT;
      GENERAL_SIGNAL : Struct
         STYLE_INIT : Bool;   // GANTRY HEARTBEAT (GANTRY TO MACHINE) / INITIATE STYLE PROGRAM
         READ_DEC_CODE : Bool;   // READ DECISION CODE
         OK_CONTINUE : Bool;   // GANTRY EMERGENCY STOP OK (GANTRY TO MACHINE) / OK TO CONTINUE
         ENTER_REQUEST : Bool;   // ENTER CELL REQUEST
         DRY_CYCLE : Bool;   // GANTRY IN MANUAL MODE (GANTRY TO MACHINE) / DRY CYCLE
         RECOVER_REQ : Bool;   // GANTRY IN AUTO MODE (GANTRY TO MACHINE) / RECOVERY REQUEST
         SPARE_68_6 : Bool;   // GANTRY IN AUTO CYCLE RUNNING (GANTRY TO MACHINE)
         SPARE_68_7 : Bool;   // GANTRY OVERHEAD DOOR CLOSED & LOCKED (GANTRY TO MACHINE)
         IMMEDIATE_STOP_AUX : Bool;
         STOP_END_OF_CYCLE : Bool;
         RUNOUT_REQUEST : Bool;
         SPARE_69_3 : Bool;
         SPARE_69_4 : Bool;
         SPARE_69_5 : Bool;
         SPARE_69_6 : Bool;
         SPARE_69_7 : Bool;
         SPARE_70_0 : Byte;   // GANTRY CLEAR OF MACHINE (GANTRY TO MACHINE)
         SPARE_71_0 : Byte;   // GANTRY CLEAR OF FIXTURE (GANTRY TO MACHINE)
         SPARE_72_0 : Byte;
         SPARE_73_0 : Byte;
      END_STRUCT;
      PROGRAM : Struct
         STYLE_PROGRAM : Byte;   // GANTRY HEARTBEAT (GANTRY TO MACHINE) / GROUP INPUT INDICATING STYLE NUMBER PROGRAM
         DEC_CODE : Byte;   // SPECIFIC OPERATING WITHIN A STYLE
         PART_TYPE : Byte;   // GANTRY EMERGENCY STOP OK (GANTRY TO MACHINE) / PART TYPE SELECTED
         SPARE_77_0 : Byte;   // GANTRY EMERGENCY STOP OK (GANTRY TO MACHINE)
      END_STRUCT;
      GRIPPERS : Struct
         T1_GRIPPER_A_OPEN_REQ : Bool;   // ROBOT TOOL 1 GRIPPER A OPEN REQUEST
         T1_GRIPPER_A_CLOSE_REQ : Bool;   // ROBOT TOOL 1 GRIPPER A CLOSE REQUEST
         SPARE_78_2 : Bool;
         SPARE_78_3 : Bool;
         T1_GRIPPER_A_OPEN : Bool;   // ROBOT TOOL 1 GRIPPER A OPEN
         T1_GRIPPER_A_CLOSED : Bool;   // ROBOT TOOL 1 GRIPPER A CLOSED
         SPARE_78_6 : Bool;
         SPARE_78_7 : Bool;
         T1_GRIPPER_B_OPEN_REQ : Bool;   // ROBOT TOOL 1 GRIPPER B OPEN REQUEST
         T1_GRIPPER_B_CLOSE_REQ : Bool;   // ROBOT TOOL 1 GRIPPER B CLOSE REQUEST
         SPARE_79_2 : Bool;
         SPARE_79_3 : Bool;
         T1_GRIPPER_B_OPEN : Bool;   // ROBOT TOOL 1 GRIPPER B OPEN
         T1_GRIPPER_B_CLOSED : Bool;   // ROBOT TOOL 1 GRIPPER B CLOSED
         SPARE_79_6 : Bool;
         SPARE_79_7 : Bool;
         T1_GRIPPER_C_OPEN_REQ : Bool;   // ROBOT TOOL 1 GRIPPER C OPEN REQUEST
         T1_GRIPPER_C_CLOSE_REQ : Bool;   // ROBOT TOOL 1 GRIPPER C CLOSE REQUEST
         SPARE_80_2 : Bool;
         SPARE_80_3 : Bool;
         T1_GRIPPER_C_OPEN : Bool;   // ROBOT TOOL 1 GRIPPER C OPEN
         T1_GRIPPER_C_CLOSED : Bool;   // ROBOT TOOL 1 GRIPPER C CLOSED
         SPARE_80_6 : Bool;
         SPARE_80_7 : Bool;
         T1_GRIPPER_D_OPEN_REQ : Bool;   // ROBOT TOOL 1 GRIPPER D OPEN REQUEST
         T1_GRIPPER_D_CLOSE_REQ : Bool;   // ROBOT TOOL 1 GRIPPER D CLOSE REQUEST
         SPARE_81_2 : Bool;
         SPARE_81_3 : Bool;
         T1_GRIPPER_D_OPEN : Bool;   // ROBOT TOOL 1 GRIPPER D OPEN
         T1_GRIPPER_D_CLOSED : Bool;   // ROBOT TOOL 1 GRIPPER D CLOSED
         SPARE_81_6 : Bool;
         SPARE_81_7 : Bool;
         T1_GRIPPER_E_OPEN_REQ : Bool;   // ROBOT TOOL 1 GRIPPER E OPEN REQUEST
         T1_GRIPPER_E_CLOSE_REQ : Bool;   // ROBOT TOOL 1 GRIPPER E CLOSE REQUEST
         SPARE_82_2 : Bool;
         SPARE_82_3 : Bool;
         T1_GRIPPER_E_OPEN : Bool;   // ROBOT TOOL 1 GRIPPER E OPEN
         T1_GRIPPER_E_CLOSED : Bool;   // ROBOT TOOL 1 GRIPPER E CLOSED
         SPARE_82_6 : Bool;
         SPARE_82_7 : Bool;
         T2_GRIPPER_A_OPEN_REQ : Bool;   // ROBOT TOOL 2 GRIPPER A OPEN REQUEST
         T2_GRIPPER_A_CLOSE_REQ : Bool;   // ROBOT TOOL 2 GRIPPER A CLOSE REQUEST
         SPARE_83_2 : Bool;
         SPARE_83_3 : Bool;
         T2_GRIPPER_A_OPEN : Bool;   // ROBOT TOOL 2 GRIPPER A OPEN
         T2_GRIPPER_A_CLOSED : Bool;   // ROBOT TOOL 2 GRIPPER A CLOSED
         SPARE_83_6 : Bool;
         SPARE_83_7 : Bool;
         T2_GRIPPER_B_OPEN_REQ : Bool;   // ROBOT TOOL 2 GRIPPER B OPEN REQUEST
         T2_GRIPPER_B_CLOSE_REQ : Bool;   // ROBOT TOOL 2 GRIPPER B CLOSE REQUEST
         SPARE_84_2 : Bool;
         SPARE_84_3 : Bool;
         T2_GRIPPER_B_OPEN : Bool;   // ROBOT TOOL 2 GRIPPER B OPEN
         T2_GRIPPER_B_CLOSED : Bool;   // ROBOT TOOL 2 GRIPPER B CLOSED
         SPARE_84_6 : Bool;
         SPARE_84_7 : Bool;
         T2_GRIPPER_C_OPEN_REQ : Bool;   // ROBOT TOOL 2 GRIPPER C OPEN REQUEST
         T2_GRIPPER_C_CLOSE_REQ : Bool;   // ROBOT TOOL 2 GRIPPER C CLOSE REQUEST
         SPARE_85_2 : Bool;
         SPARE_85_3 : Bool;
         T2_GRIPPER_C_OPEN : Bool;   // ROBOT TOOL 2 GRIPPER C OPEN
         T2_GRIPPER_C_CLOSED : Bool;   // ROBOT TOOL 2 GRIPPER C CLOSED
         SPARE_85_6 : Bool;
         SPARE_85_7 : Bool;
         T2_GRIPPER_D_OPEN_REQ : Bool;   // ROBOT TOOL 2 GRIPPER D OPEN REQUEST
         T2_GRIPPER_D_CLOSE_REQ : Bool;   // ROBOT TOOL 2 GRIPPER D CLOSE REQUEST
         SPARE_86_2 : Bool;
         SPARE_86_3 : Bool;
         T2_GRIPPER_D_OPEN : Bool;   // ROBOT TOOL 2 GRIPPER D OPEN
         T2_GRIPPER_D_CLOSED : Bool;   // ROBOT TOOL 2 GRIPPER D CLOSED
         SPARE_86_6 : Bool;
         SPARE_86_7 : Bool;
         T2_GRIPPER_E_OPEN_REQ : Bool;   // ROBOT TOOL 2 GRIPPER E OPEN REQUEST
         T2_GRIPPER_E_CLOSE_REQ : Bool;   // ROBOT TOOL 2 GRIPPER E CLOSE REQUEST
         SPARE_87_2 : Bool;
         SPARE_87_3 : Bool;
         T2_GRIPPER_E_OPEN : Bool;   // ROBOT TOOL 2 GRIPPER E OPEN
         T2_GRIPPER_E_CLOSED : Bool;   // ROBOT TOOL 2 GRIPPER E CLOSED
         SPARE_87_6 : Bool;
         SPARE_87_7 : Bool;
         T1_ALL_GRIPS_OPEN_REQ : Bool;   // ROBOT TOOL 1 OPEN ALL GRIPPERS REQUEST
         T1_ALL_GRIPS_CLOSE_REQ : Bool;   // ROBOT TOOL 1 CLOSE ALL GRIPPERS REQUEST
         T1_ALL_GRIPPERS_OPEN : Bool;   // ROBOT TOOL 1 ALL GRIPPERS OPEN
         T1_ALL_GRIPPERS_CLOSED : Bool;   // ROBOT TOOL 1 ALL GRIPPERS CLOSED
         SPARE_88_4 : Bool;
         SPARE_88_5 : Bool;
         SPARE_88_6 : Bool;
         SPARE_88_7 : Bool;
         T2_ALL_GRIPS_OPEN_REQ : Bool;   // ROBOT TOOL 2 CLOSE ALL GRIPPERS REQUEST
         T2_ALL_GRIPS_CLOSE_REQ : Bool;   // ROBOT TOOL 2 CLOSE ALL GRIPPERS REQUEST
         T2_ALL_GRIPPERS_OPEN : Bool;   // ROBOT TOOL 2 ALL GRIPPERS OPEN
         T2_ALL_GRIPPERS_CLOSED : Bool;   // ROBOT TOOL 2 ALL GRIPPERS CLOSED
         SPARE_89_4 : Bool;
         SPARE_89_5 : Bool;
         SPARE_89_6 : Bool;
         SPARE_89_7 : Bool;
         SPARE_90_0 : Byte;
         FAULT_NUMBER : Byte;   // FAULT RESPONSE
      END_STRUCT;
      CLEARS : Struct
         CLEAR_U_1 : Bool;   // GANTRY HEARTBEAT (GANTRY TO MACHINE) / CLEAR TO GET IN UNIT 1
         CLEAR_U_2 : Bool;   // CLEAR TO GET IN UNIT 2
         CLEAR_U_3 : Bool;   // GANTRY EMERGENCY STOP OK (GANTRY TO MACHINE) / CLEAR TO GET IN UNIT 3
         CLEAR_U_4 : Bool;   // CLEAR TO GET IN UNIT 4
         CLEAR_U_5 : Bool;   // GANTRY IN MANUAL MODE (GANTRY TO MACHINE) / CLEAR TO GET IN UNIT 5
         CLEAR_U_6 : Bool;   // GANTRY IN AUTO MODE (GANTRY TO MACHINE) / CLEAR TO GET IN UNIT 6
         CLEAR_U_7 : Bool;   // GANTRY IN AUTO CYCLE RUNNING (GANTRY TO MACHINE) / CLEAR TO GET IN UNIT 7
         CLEAR_U_8 : Bool;   // GANTRY OVERHEAD DOOR CLOSED & LOCKED (GANTRY TO MACHINE) / CLEAR TO GET IN UNIT 8
         CLEAR_U_9 : Bool;   // GANTRY IN RUN OUT COMPLETE(GANTRY TO MACHINE) / CLEAR TO GET IN UNIT 9
         CLEAR_U_10 : Bool;   // GANTRY CLEAR OF MACHINE (GANTRY TO MACHINE) / CLEAR TO GET IN UNIT 10
         SPARE_93_2 : Bool;   // GANTRY CLEAR OF FIXTURE (GANTRY TO MACHINE)
         SPARE_93_3 : Bool;
         SPARE_93_4 : Bool;
         SPARE_93_5 : Bool;   // GANTRY PART TYPE CHANGE REQUESTED (GANTRY TO MACHINE)
         SPARE_93_6 : Bool;   // GANTRY REQUEST MACHINE TO RUN WITH LOADED PARTS (GANTRY TO MACHINE)
         SPARE_93_7 : Bool;   // GANTRY RUN OUT REQUESTED (GANTRY TO MACHINE)
         SPARE_94_0 : Byte;
         SPARE_95_0 : Byte;
      END_STRUCT;
      TASKS : Struct
         COMPLETE_TSK_1 : Bool;   // GANTRY HEARTBEAT (GANTRY TO MACHINE) / PICK REQUEST - ST1
         COMPLETE_TSK_2 : Bool;   // PLACE REQUEST - ST1
         COMPLETE_TSK_3 : Bool;   // GANTRY EMERGENCY STOP OK (GANTRY TO MACHINE) / PICK&PLACE REQUEST - ST1
         COMPLETE_TSK_4 : Bool;   // ROBOT COMPLETE TASK 4
         COMPLETE_TSK_5 : Bool;   // GANTRY IN MANUAL MODE (GANTRY TO MACHINE) / ROBOT COMPLETE TASK 5
         COMPLETE_TSK_6 : Bool;   // GANTRY IN AUTO MODE (GANTRY TO MACHINE) / ROBOT COMPLETE TASK 6
         COMPLETE_TSK_7 : Bool;   // GANTRY IN AUTO CYCLE RUNNING (GANTRY TO MACHINE) / ROBOT COMPLETE TASK 7
         COMPLETE_TSK_8 : Bool;   // GANTRY OVERHEAD DOOR CLOSED & LOCKED (GANTRY TO MACHINE) / ROBOT COMPLETE TASK 8
         SPARE_97_0 : Byte;   // GANTRY IN RUN OUT COMPLETE(GANTRY TO MACHINE)
         SPARE_98_0 : Byte;   // GANTRY CLEAR OF MACHINE (GANTRY TO MACHINE)
         SPARE_99_0 : Byte;   // GANTRY CLEAR OF FIXTURE (GANTRY TO MACHINE)
         SPARE_100_0 : Byte;
         SPARE_101_0 : Byte;
         SPARE_102_0 : Byte;
         SPARE_103_0 : Byte;
      END_STRUCT;
      PARTS_ENABLED : Struct
         PART_A_ENABLED : Bool;   // GANTRY HEARTBEAT (GANTRY TO MACHINE) / PART A ENABLED TO WORK
         PART_B_ENABLED : Bool;   // PART B ENABLED TO WORK
         PART_C_ENABLED : Bool;   // GANTRY EMERGENCY STOP OK (GANTRY TO MACHINE) / PART C ENABLED TO WORK
         PART_D_ENABLED : Bool;   // PART D ENABLED TO WORK
         PART_E_ENABLED : Bool;   // GANTRY IN MANUAL MODE (GANTRY TO MACHINE) / PART E ENABLED TO WORK
         SPARE_104_5 : Bool;   // GANTRY IN AUTO MODE (GANTRY TO MACHINE)
         SPARE_104_6 : Bool;   // GANTRY IN AUTO CYCLE RUNNING (GANTRY TO MACHINE)
         SPARE_104_7 : Bool;   // GANTRY OVERHEAD DOOR CLOSED & LOCKED (GANTRY TO MACHINE)
         SPARE_105_0 : Byte;   // GANTRY CLEAR OF FIXTURE (GANTRY TO MACHINE)
      END_STRUCT;
      SPARES : Array[106..127] of Byte;
   END_STRUCT;
END_TYPE

